LIN {X 0,Y 467.704,Z 292.228,A -85,B 0,C 180,E1 -7476.035,E2 -7476.035} C_VEL
LIN {X 0,Y 467.665,Z 292.229,A -85,B 0,C 180,E1 -7478.64,E2 -7478.64} C_VEL
LIN {X 0,Y 467.684,Z 292.329,A -85,B 0,C 180,E1 -7481.125,E2 -7481.125} C_VEL
LIN {X 0,Y 468.727,Z 299.708,A -85,B 0,C 180,E1 -7482.725,E2 -7482.725} C_VEL
LIN {X 0,Y 468.456,Z 310.96,A -85,B 0,C 180,E1 -7485.05,E2 -7485.05} C_VEL
LIN {X 0,Y 471.306,Z 325.447,A -85,B 0,C 180,E1 -7485.4,E2 -7485.4} C_VEL
LIN {X 0,Y 470.52,Z 418.247,A -85,B 0,C 180,E1 -7486.862,E2 -7486.862} C_VEL
LIN {X 0,Y 470.256,Z 431.761,A -85,B 0,C 180,E1 -7487.255,E2 -7487.255} C_VEL
LIN {X 0,Y 469.928,Z 444.22,A -85,B 0,C 180,E1 -7487.793,E2 -7487.793} C_VEL
LIN {X 0,Y 469.506,Z 455.23,A -85,B 0,C 180,E1 -7488.43,E2 -7488.43} C_VEL
LIN {X 0,Y 469.027,Z 466.456,A -85,B 0,C 180,E1 -7489.264,E2 -7489.264} C_VEL
LIN {X 0,Y 468.47,Z 477.517,A -85,B 0,C 180,E1 -7490.295,E2 -7490.295} C_VEL
LIN {X 0,Y 468.012,Z 487.034,A -85,B 0,C 180,E1 -7491.402,E2 -7491.402} C_VEL
LIN {X 0,Y 467.679,Z 494.909,A -85,B 0,C 180,E1 -7492.527,E2 -7492.527} C_VEL
LIN {X 0,Y 467.319,Z 502.972,A -85,B 0,C 180,E1 -7493.952,E2 -7493.952} C_VEL
LIN {X 0,Y 467.082,Z 508.521,A -85,B 0,C 180,E1 -7495.183,E2 -7495.183} C_VEL
LIN {X 0,Y 466.913,Z 512.769,A -85,B 0,C 180,E1 -7496.357,E2 -7496.357} C_VEL
LIN {X 0,Y 466.762,Z 516.837,A -85,B 0,C 180,E1 -7497.819,E2 -7497.819} C_VEL
LIN {X 0,Y 466.632,Z 519.377,A -85,B 0,C 180,E1 -7499.126,E2 -7499.126} C_VEL
LIN {X 0,Y 466.562,Z 521.275,A -85,B 0,C 180,E1 -7500.838,E2 -7500.838} C_VEL
LIN {X 0,Y 466.549,Z 521.623,A -85,B 0,C 180,E1 -7502.48,E2 -7502.48} C_VEL
LIN {X 0,Y 466.552,Z 520.636,A -85,B 0,C 180,E1 -7504.054,E2 -7504.054} C_VEL
LIN {X 0,Y 466.699,Z 518.356,A -85,B 0,C 180,E1 -7505.591,E2 -7505.591} C_VEL
LIN {X 0,Y 466.821,Z 514.889,A -85,B 0,C 180,E1 -7507.068,E2 -7507.068} C_VEL
LIN {X 0,Y 467.024,Z 510.213,A -85,B 0,C 180,E1 -7508.508,E2 -7508.508} C_VEL
LIN {X 0,Y 467.265,Z 504.294,A -85,B 0,C 180,E1 -7509.908,E2 -7509.908} C_VEL
LIN {X 0,Y 467.591,Z 496.918,A -85,B 0,C 180,E1 -7511.278,E2 -7511.278} C_VEL
LIN {X 0,Y 468.015,Z 488.675,A -85,B 0,C 180,E1 -7512.505,E2 -7512.505} C_VEL
LIN {X 0,Y 468.474,Z 479.399,A -85,B 0,C 180,E1 -7513.629,E2 -7513.629} C_VEL
LIN {X 0,Y 468.998,Z 468.987,A -85,B 0,C 180,E1 -7514.648,E2 -7514.648} C_VEL
LIN {X 0,Y 469.505,Z 457.587,A -85,B 0,C 180,E1 -7515.532,E2 -7515.532} C_VEL
LIN {X 0,Y 469.927,Z 445.273,A -85,B 0,C 180,E1 -7516.277,E2 -7516.277} C_VEL
LIN {X 0,Y 470.301,Z 432.788,A -85,B 0,C 180,E1 -7516.829,E2 -7516.829} C_VEL
LIN {X 0,Y 470.561,Z 419.847,A -85,B 0,C 180,E1 -7517.218,E2 -7517.218} C_VEL
LIN {X 0,Y 470.874,Z 388.179,A -85,B 0,C 180,E1 -7517.741,E2 -7517.741} C_VEL
LIN {X 0,Y 471.357,Z 325.273,A -85,B 0,C 180,E1 -7518.725,E2 -7518.725} C_VEL
LIN {X 0,Y 468.506,Z 310.615,A -85,B 0,C 180,E1 -7519.089,E2 -7519.089} C_VEL
LIN {X 0,Y 468.614,Z 298.408,A -85,B 0,C 180,E1 -7521.344,E2 -7521.344} C_VEL
LIN {X 0,Y 467.552,Z 292.248,A -85,B 0,C 180,E1 -7522.545,E2 -7522.545} C_VEL
LIN {X 0,Y 467.55,Z 292.246,A -85,B 0,C 180,E1 -7525.754,E2 -7525.754} C_VEL
LIN {X 0,Y 467.529,Z 292.247,A -85,B 0,C 180,E1 -7528.951,E2 -7528.951} C_VEL
LIN {X 0,Y 467.601,Z 292.244,A -85,B 0,C 180,E1 -7532.456,E2 -7532.456} C_VEL
LIN {X 0,Y 467.557,Z 292.245,A -85,B 0,C 180,E1 -7535.11,E2 -7535.11} C_VEL
LIN {X 0,Y 467.485,Z 292.255,A -85,B 0,C 180,E1 -7537.924,E2 -7537.924} C_VEL
LIN {X 0,Y 467.573,Z 292.244,A -85,B 0,C 180,E1 -7540.69,E2 -7540.69} C_VEL
LIN {X 0,Y 467.597,Z 292.237,A -85,B 0,C 180,E1 -7544.113,E2 -7544.113} C_VEL
LIN {X 0,Y 467.601,Z 292.235,A -85,B 0,C 180,E1 -7547.641,E2 -7547.641} C_VEL
LIN {X 0,Y 467.613,Z 292.236,A -85,B 0,C 180,E1 -7550.484,E2 -7550.484} C_VEL
LIN {X 0,Y 467.646,Z 292.232,A -85,B 0,C 180,E1 -7553.095,E2 -7553.095} C_VEL
LIN {X 0,Y 467.67,Z 292.231,A -85,B 0,C 180,E1 -7554.827,E2 -7554.827} C_VEL
LIN {X 0,Y 467.811,Z 292.209,A -85,B 0,C 180,E1 -7557.417,E2 -7557.417} C_VEL
LIN {X 0,Y 467.776,Z 292.217,A -85,B 0,C 180,E1 -7560.861,E2 -7560.861} C_VEL
LIN {X 0,Y 467.813,Z 292.212,A -85,B 0,C 180,E1 -7562.583,E2 -7562.583} C_VEL
LIN {X 0,Y 467.699,Z 292.222,A -85,B 0,C 180,E1 -7566.038,E2 -7566.038} C_VEL
LIN {X 0,Y 467.636,Z 292.229,A -85,B 0,C 180,E1 -7568.644,E2 -7568.644} C_VEL
LIN {X 0,Y 467.646,Z 292.224,A -85,B 0,C 180,E1 -7572.146,E2 -7572.146} C_VEL
LIN {X 0,Y 467.617,Z 292.228,A -85,B 0,C 180,E1 -7575.895,E2 -7575.895} C_VEL
LIN {X 0,Y 467.575,Z 292.24,A -85,B 0,C 180,E1 -7579.31,E2 -7579.31} C_VEL
LIN {X 0,Y 467.532,Z 292.242,A -85,B 0,C 180,E1 -7582.074,E2 -7582.074} C_VEL
LIN {X 0,Y 467.575,Z 292.235,A -85,B 0,C 180,E1 -7584.889,E2 -7584.889} C_VEL
LIN {X 0,Y 467.584,Z 292.236,A -85,B 0,C 180,E1 -7587.771,E2 -7587.771} C_VEL
LIN {X 0,Y 467.531,Z 292.246,A -85,B 0,C 180,E1 -7591.049,E2 -7591.049} C_VEL
LIN {X 0,Y 467.55,Z 292.24,A -85,B 0,C 180,E1 -7594.246,E2 -7594.246} C_VEL
LIN {X 0,Y 467.524,Z 292.248,A -85,B 0,C 180,E1 -7597.192,E2 -7597.192} C_VEL
LIN {X 0,Y 467.579,Z 292.241,A -85,B 0,C 180,E1 -7599.963,E2 -7599.963} C_VEL
LIN {X 0,Y 467.586,Z 292.239,A -85,B 0,C 180,E1 -7602.575,E2 -7602.575} C_VEL
LIN {X 0,Y 467.544,Z 292.247,A -85,B 0,C 180,E1 -7606.181,E2 -7606.181} C_VEL
LIN {X 0,Y 467.563,Z 292.241,A -85,B 0,C 180,E1 -7608.726,E2 -7608.726} C_VEL
LIN {X 0,Y 467.555,Z 292.245,A -85,B 0,C 180,E1 -7611.411,E2 -7611.411} C_VEL
LIN {X 0,Y 467.541,Z 292.247,A -85,B 0,C 180,E1 -7614.264,E2 -7614.264} C_VEL
LIN {X 0,Y 467.563,Z 292.245,A -85,B 0,C 180,E1 -7617.325,E2 -7617.325} C_VEL
LIN {X 0,Y 467.562,Z 292.245,A -85,B 0,C 180,E1 -7620.67,E2 -7620.67} C_VEL
LIN {X 0,Y 467.614,Z 292.24,A -85,B 0,C 180,E1 -7623.686,E2 -7623.686} C_VEL
LIN {X 0,Y 467.64,Z 292.332,A -85,B 0,C 180,E1 -7624.137,E2 -7624.137} C_VEL
LIN {X 0,Y 469.709,Z 303.354,A -85,B 0,C 180,E1 -7626.177,E2 -7626.177} C_VEL
LIN {X 0,Y 469.179,Z 319.417,A -85,B 0,C 180,E1 -7628.935,E2 -7628.935} C_VEL
LIN {X 0,Y 468.465,Z 338.052,A -85,B 0,C 180,E1 -7632.093,E2 -7632.093} C_VEL
LIN {X 0,Y 468.269,Z 343.322,A -85,B 0,C 180,E1 -7632.962,E2 -7632.962} C_VEL
LIN {X 0,Y 471.212,Z 363.176,A -85,B 0,C 180,E1 -7633.389,E2 -7633.389} C_VEL
LIN {X 0,Y 470.443,Z 452.18,A -85,B 0,C 180,E1 -7634.793,E2 -7634.793} C_VEL
LIN {X 0,Y 470.061,Z 466.055,A -85,B 0,C 180,E1 -7635.196,E2 -7635.196} C_VEL
LIN {X 0,Y 469.561,Z 479.027,A -85,B 0,C 180,E1 -7635.762,E2 -7635.762} C_VEL
LIN {X 0,Y 469.134,Z 490.835,A -85,B 0,C 180,E1 -7636.467,E2 -7636.467} C_VEL
LIN {X 0,Y 468.58,Z 502.825,A -85,B 0,C 180,E1 -7637.383,E2 -7637.383} C_VEL
LIN {X 0,Y 468.157,Z 512.507,A -85,B 0,C 180,E1 -7638.311,E2 -7638.311} C_VEL
LIN {X 0,Y 467.69,Z 521.747,A -85,B 0,C 180,E1 -7639.396,E2 -7639.396} C_VEL
LIN {X 0,Y 467.274,Z 530.751,A -85,B 0,C 180,E1 -7640.699,E2 -7640.699} C_VEL
LIN {X 0,Y 467.006,Z 538.009,A -85,B 0,C 180,E1 -7642.002,E2 -7642.002} C_VEL
LIN {X 0,Y 466.851,Z 542.909,A -85,B 0,C 180,E1 -7643.086,E2 -7643.086} C_VEL
LIN {X 0,Y 466.76,Z 547.675,A -85,B 0,C 180,E1 -7644.387,E2 -7644.387} C_VEL
LIN {X 0,Y 466.646,Z 551.315,A -85,B 0,C 180,E1 -7645.684,E2 -7645.684} C_VEL
LIN {X 0,Y 466.689,Z 553.198,A -85,B 0,C 180,E1 -7646.55,E2 -7646.55} C_VEL
LIN {X 0,Y 466.661,Z 554.607,A -85,B 0,C 180,E1 -7647.413,E2 -7647.413} C_VEL
LIN {X 0,Y 466.619,Z 556.232,A -85,B 0,C 180,E1 -7649.14,E2 -7649.14} C_VEL
LIN {X 0,Y 466.6,Z 556.451,A -85,B 0,C 180,E1 -7650.003,E2 -7650.003} C_VEL
LIN {X 0,Y 466.619,Z 556.236,A -85,B 0,C 180,E1 -7650.866,E2 -7650.866} C_VEL
LIN {X 0,Y 466.662,Z 554.629,A -85,B 0,C 180,E1 -7652.592,E2 -7652.592} C_VEL
LIN {X 0,Y 466.69,Z 553.223,A -85,B 0,C 180,E1 -7653.456,E2 -7653.456} C_VEL
LIN {X 0,Y 466.69,Z 550.267,A -85,B 0,C 180,E1 -7654.753,E2 -7654.753} C_VEL
LIN {X 0,Y 466.752,Z 546.264,A -85,B 0,C 180,E1 -7656.053,E2 -7656.053} C_VEL
LIN {X 0,Y 466.943,Z 540.102,A -85,B 0,C 180,E1 -7657.57,E2 -7657.57} C_VEL
LIN {X 0,Y 467.167,Z 533.373,A -85,B 0,C 180,E1 -7658.873,E2 -7658.873} C_VEL
LIN {X 0,Y 467.505,Z 525.026,A -85,B 0,C 180,E1 -7660.176,E2 -7660.176} C_VEL
LIN {X 0,Y 467.954,Z 516.447,A -85,B 0,C 180,E1 -7661.261,E2 -7661.261} C_VEL
LIN {X 0,Y 468.472,Z 506.349,A -85,B 0,C 180,E1 -7662.3,E2 -7662.3} C_VEL
LIN {X 0,Y 468.906,Z 495.369,A -85,B 0,C 180,E1 -7663.215,E2 -7663.215} C_VEL
LIN {X 0,Y 469.392,Z 483.818,A -85,B 0,C 180,E1 -7663.973,E2 -7663.973} C_VEL
LIN {X 0,Y 469.832,Z 471.84,A -85,B 0,C 180,E1 -7664.568,E2 -7664.568} C_VEL
LIN {X 0,Y 470.277,Z 458.915,A -85,B 0,C 180,E1 -7665.024,E2 -7665.024} C_VEL
LIN {X 0,Y 470.546,Z 445.237,A -85,B 0,C 180,E1 -7665.32,E2 -7665.32} C_VEL
LIN {X 0,Y 471.139,Z 362.545,A -85,B 0,C 180,E1 -7666.605,E2 -7666.605} C_VEL
LIN {X 0,Y 468.314,Z 343.69,A -85,B 0,C 180,E1 -7667.018,E2 -7667.018} C_VEL
LIN {X 0,Y 469.052,Z 325.465,A -85,B 0,C 180,E1 -7670.16,E2 -7670.16} C_VEL
LIN {X 0,Y 469.878,Z 307.217,A -85,B 0,C 180,E1 -7673.352,E2 -7673.352} C_VEL
LIN {X 0,Y 469.713,Z 302.985,A -85,B 0,C 180,E1 -7674.118,E2 -7674.118} C_VEL
LIN {X 0,Y 467.659,Z 292.234,A -85,B 0,C 180,E1 -7676.197,E2 -7676.197} C_VEL
LIN {X 0,Y 467.573,Z 292.242,A -85,B 0,C 180,E1 -7679.333,E2 -7679.333} C_VEL
LIN {X 0,Y 467.585,Z 292.237,A -85,B 0,C 180,E1 -7682.679,E2 -7682.679} C_VEL
LIN {X 0,Y 467.563,Z 292.241,A -85,B 0,C 180,E1 -7685.739,E2 -7685.739} C_VEL
LIN {X 0,Y 467.562,Z 292.238,A -85,B 0,C 180,E1 -7689.147,E2 -7689.147} C_VEL
LIN {X 0,Y 467.588,Z 292.241,A -85,B 0,C 180,E1 -7692.567,E2 -7692.567} C_VEL
LIN {X 0,Y 467.566,Z 292.239,A -85,B 0,C 180,E1 -7695.052,E2 -7695.052} C_VEL
LIN {X 0,Y 467.589,Z 292.235,A -85,B 0,C 180,E1 -7697.44,E2 -7697.44} C_VEL
LIN {X 0,Y 467.58,Z 292.24,A -85,B 0,C 180,E1 -7700.855,E2 -7700.855} C_VEL
LIN {X 0,Y 467.559,Z 292.242,A -85,B 0,C 180,E1 -7704.26,E2 -7704.26} C_VEL
LIN {X 0,Y 467.579,Z 292.237,A -85,B 0,C 180,E1 -7707.321,E2 -7707.321} C_VEL
LIN {X 0,Y 467.567,Z 292.245,A -85,B 0,C 180,E1 -7710.667,E2 -7710.667} C_VEL
LIN {X 0,Y 467.611,Z 292.236,A -85,B 0,C 180,E1 -7713.199,E2 -7713.199} C_VEL
LIN {X 0,Y 467.587,Z 292.238,A -85,B 0,C 180,E1 -7716.468,E2 -7716.468} C_VEL
LIN {X 0,Y 467.615,Z 292.232,A -85,B 0,C 180,E1 -7719.777,E2 -7719.777} C_VEL
LIN {X 0,Y 467.598,Z 292.235,A -85,B 0,C 180,E1 -7722.506,E2 -7722.506} C_VEL
LIN {X 0,Y 467.597,Z 292.242,A -85,B 0,C 180,E1 -7725.196,E2 -7725.196} C_VEL
LIN {X 0,Y 467.647,Z 292.229,A -85,B 0,C 180,E1 -7727.854,E2 -7727.854} C_VEL
LIN {X 0,Y 467.672,Z 292.232,A -85,B 0,C 180,E1 -7731.357,E2 -7731.357} C_VEL
LIN {X 0,Y 467.723,Z 292.219,A -85,B 0,C 180,E1 -7733.962,E2 -7733.962} C_VEL
LIN {X 0,Y 467.847,Z 292.212,A -85,B 0,C 180,E1 -7737.417,E2 -7737.417} C_VEL
LIN {X 0,Y 467.866,Z 292.202,A -85,B 0,C 180,E1 -7740,E2 -7740} C_VEL
LIN {X 0,Y 467.846,Z 292.203,A -85,B 0,C 180,E1 -7742.583,E2 -7742.583} C_VEL
LIN {X 0,Y 467.708,Z 292.223,A -85,B 0,C 180,E1 -7746.038,E2 -7746.038} C_VEL
LIN {X 0,Y 467.659,Z 292.226,A -85,B 0,C 180,E1 -7748.643,E2 -7748.643} C_VEL
LIN {X 0,Y 467.646,Z 292.231,A -85,B 0,C 180,E1 -7752.146,E2 -7752.146} C_VEL
LIN {X 0,Y 467.64,Z 292.237,A -85,B 0,C 180,E1 -7755.884,E2 -7755.884} C_VEL
LIN {X 0,Y 467.612,Z 292.233,A -85,B 0,C 180,E1 -7759.308,E2 -7759.308} C_VEL
LIN {X 0,Y 467.522,Z 292.251,A -85,B 0,C 180,E1 -7762.075,E2 -7762.075} C_VEL
LIN {X 0,Y 467.548,Z 292.24,A -85,B 0,C 180,E1 -7764.891,E2 -7764.891} C_VEL
LIN {X 0,Y 467.537,Z 292.245,A -85,B 0,C 180,E1 -7767.774,E2 -7767.774} C_VEL
LIN {X 0,Y 467.543,Z 292.241,A -85,B 0,C 180,E1 -7771.041,E2 -7771.041} C_VEL
LIN {X 0,Y 467.571,Z 292.245,A -85,B 0,C 180,E1 -7774.24,E2 -7774.24} C_VEL
LIN {X 0,Y 467.51,Z 292.245,A -85,B 0,C 180,E1 -7777.181,E2 -7777.181} C_VEL
LIN {X 0,Y 467.535,Z 292.248,A -85,B 0,C 180,E1 -7780.269,E2 -7780.269} C_VEL
LIN {X 0,Y 467.515,Z 292.252,A -85,B 0,C 180,E1 -7782.569,E2 -7782.569} C_VEL
LIN {X 0,Y 467.552,Z 292.242,A -85,B 0,C 180,E1 -7785.051,E2 -7785.051} C_VEL
LIN {X 0,Y 467.55,Z 292.247,A -85,B 0,C 180,E1 -7788.727,E2 -7788.727} C_VEL
LIN {X 0,Y 467.532,Z 292.242,A -85,B 0,C 180,E1 -7791.952,E2 -7791.952} C_VEL
LIN {X 0,Y 467.489,Z 292.251,A -85,B 0,C 180,E1 -7795.16,E2 -7795.16} C_VEL
LIN {X 0,Y 467.543,Z 292.242,A -85,B 0,C 180,E1 -7798.256,E2 -7798.256} C_VEL
LIN {X 0,Y 467.528,Z 292.247,A -85,B 0,C 180,E1 -7801.246,E2 -7801.246} C_VEL
LIN {X 0,Y 467.563,Z 292.239,A -85,B 0,C 180,E1 -7804.405,E2 -7804.405} C_VEL
LIN {X 0,Y 467.577,Z 292.244,A -85,B 0,C 180,E1 -7806.995,E2 -7806.995} C_VEL
LIN {X 0,Y 467.623,Z 292.232,A -85,B 0,C 180,E1 -7809.776,E2 -7809.776} C_VEL
LIN {X 0,Y 467.589,Z 292.235,A -85,B 0,C 180,E1 -7812.504,E2 -7812.504} C_VEL
LIN {X 0,Y 467.594,Z 292.239,A -85,B 0,C 180,E1 -7815.403,E2 -7815.403} C_VEL
LIN {X 0,Y 466.923,Z 292.32,A -85,B 0,C 180,E1 -7816.123,E2 -7816.123} C_VEL
LIN {X 0,Y 464.083,Z 292.68,A -85,B 0,C 180,E1 -7817.291,E2 -7817.291} C_VEL
LIN {X 0,Y 461.685,Z 292.974,A -85,B 0,C 180,E1 -7818.233,E2 -7818.233} C_VEL
LIN {X 0,Y 460.655,Z 293.102,A -85,B 0,C 180,E1 -7818.961,E2 -7818.961} C_VEL
LIN {X 0,Y 460.57,Z 293.114,A -85,B 0,C 180,E1 -7819.208,E2 -7819.208} C_VEL
LIN {X 0,Y 460.668,Z 293.097,A -85,B 0,C 180,E1 -7822.591,E2 -7822.591} C_VEL
LIN {X 0,Y 460.678,Z 293.096,A -85,B 0,C 180,E1 -7824.746,E2 -7824.746} C_VEL
LIN {X 0,Y 460.759,Z 293.091,A -85,B 0,C 180,E1 -7827.375,E2 -7827.375} C_VEL
LIN {X 0,Y 460.821,Z 293.081,A -85,B 0,C 180,E1 -7829.997,E2 -7829.997} C_VEL
LIN {X 0,Y 460.76,Z 293.085,A -85,B 0,C 180,E1 -7832.62,E2 -7832.62} C_VEL
LIN {X 0,Y 460.669,Z 293.103,A -85,B 0,C 180,E1 -7836.127,E2 -7836.127} C_VEL
LIN {X 0,Y 460.615,Z 293.107,A -85,B 0,C 180,E1 -7838.773,E2 -7838.773} C_VEL
LIN {X 0,Y 460.613,Z 293.147,A -85,B 0,C 180,E1 -7840.936,E2 -7840.936} C_VEL
LIN {X 0,Y 461.761,Z 300.65,A -85,B 0,C 180,E1 -7842.59,E2 -7842.59} C_VEL
LIN {X 0,Y 461.491,Z 311.259,A -85,B 0,C 180,E1 -7844.803,E2 -7844.803} C_VEL
LIN {X 0,Y 464.534,Z 327.145,A -85,B 0,C 180,E1 -7845.18,E2 -7845.18} C_VEL
LIN {X 0,Y 463.635,Z 418.904,A -85,B 0,C 180,E1 -7846.65,E2 -7846.65} C_VEL
LIN {X 0,Y 463.391,Z 432.539,A -85,B 0,C 180,E1 -7847.059,E2 -7847.059} C_VEL
LIN {X 0,Y 463.054,Z 444.473,A -85,B 0,C 180,E1 -7847.586,E2 -7847.586} C_VEL
LIN {X 0,Y 462.588,Z 455.843,A -85,B 0,C 180,E1 -7848.257,E2 -7848.257} C_VEL
LIN {X 0,Y 462.039,Z 467.632,A -85,B 0,C 180,E1 -7849.156,E2 -7849.156} C_VEL
LIN {X 0,Y 461.497,Z 478.025,A -85,B 0,C 180,E1 -7850.15,E2 -7850.15} C_VEL
LIN {X 0,Y 461.037,Z 487.092,A -85,B 0,C 180,E1 -7851.221,E2 -7851.221} C_VEL
LIN {X 0,Y 460.665,Z 495.329,A -85,B 0,C 180,E1 -7852.416,E2 -7852.416} C_VEL
LIN {X 0,Y 460.328,Z 502.267,A -85,B 0,C 180,E1 -7853.645,E2 -7853.645} C_VEL
LIN {X 0,Y 460.043,Z 507.767,A -85,B 0,C 180,E1 -7854.837,E2 -7854.837} C_VEL
LIN {X 0,Y 459.857,Z 513.12,A -85,B 0,C 180,E1 -7856.304,E2 -7856.304} C_VEL
LIN {X 0,Y 459.683,Z 516.546,A -85,B 0,C 180,E1 -7857.532,E2 -7857.532} C_VEL
LIN {X 0,Y 459.595,Z 518.224,A -85,B 0,C 180,E1 -7858.292,E2 -7858.292} C_VEL
LIN {X 0,Y 459.521,Z 520.017,A -85,B 0,C 180,E1 -7859.335,E2 -7859.335} C_VEL
LIN {X 0,Y 459.45,Z 521.671,A -85,B 0,C 180,E1 -7861.062,E2 -7861.062} C_VEL
LIN {X 0,Y 459.437,Z 521.849,A -85,B 0,C 180,E1 -7862.718,E2 -7862.718} C_VEL
LIN {X 0,Y 459.481,Z 520.459,A -85,B 0,C 180,E1 -7864.461,E2 -7864.461} C_VEL
LIN {X 0,Y 459.647,Z 518.184,A -85,B 0,C 180,E1 -7865.868,E2 -7865.868} C_VEL
LIN {X 0,Y 459.775,Z 514.575,A -85,B 0,C 180,E1 -7867.358,E2 -7867.358} C_VEL
LIN {X 0,Y 460.026,Z 509.729,A -85,B 0,C 180,E1 -7868.817,E2 -7868.817} C_VEL
LIN {X 0,Y 460.261,Z 503.628,A -85,B 0,C 180,E1 -7870.228,E2 -7870.228} C_VEL
LIN {X 0,Y 460.634,Z 496.009,A -85,B 0,C 180,E1 -7871.616,E2 -7871.616} C_VEL
LIN {X 0,Y 461.126,Z 487.15,A -85,B 0,C 180,E1 -7872.912,E2 -7872.912} C_VEL
LIN {X 0,Y 461.667,Z 477.05,A -85,B 0,C 180,E1 -7874.089,E2 -7874.089} C_VEL
LIN {X 0,Y 462.21,Z 465.78,A -85,B 0,C 180,E1 -7875.141,E2 -7875.141} C_VEL
LIN {X 0,Y 462.718,Z 454.964,A -85,B 0,C 180,E1 -7875.938,E2 -7875.938} C_VEL
LIN {X 0,Y 463.137,Z 443.723,A -85,B 0,C 180,E1 -7876.586,E2 -7876.586} C_VEL
LIN {X 0,Y 463.558,Z 430.282,A -85,B 0,C 180,E1 -7877.154,E2 -7877.154} C_VEL
LIN {X 0,Y 463.804,Z 417.667,A -85,B 0,C 180,E1 -7877.506,E2 -7877.506} C_VEL
LIN {X 0,Y 464.631,Z 326.727,A -85,B 0,C 180,E1 -7878.962,E2 -7878.962} C_VEL
LIN {X 0,Y 461.585,Z 310.91,A -85,B 0,C 180,E1 -7879.352,E2 -7879.352} C_VEL
LIN {X 0,Y 461.605,Z 298.605,A -85,B 0,C 180,E1 -7881.653,E2 -7881.653} C_VEL
LIN {X 0,Y 460.532,Z 293.121,A -85,B 0,C 180,E1 -7882.774,E2 -7882.774} C_VEL
LIN {X 0,Y 460.509,Z 293.123,A -85,B 0,C 180,E1 -7885.62,E2 -7885.62} C_VEL
LIN {X 0,Y 460.495,Z 293.125,A -85,B 0,C 180,E1 -7888.741,E2 -7888.741} C_VEL
LIN {X 0,Y 460.545,Z 293.123,A -85,B 0,C 180,E1 -7892.249,E2 -7892.249} C_VEL
LIN {X 0,Y 460.513,Z 293.126,A -85,B 0,C 180,E1 -7894.703,E2 -7894.703} C_VEL
LIN {X 0,Y 460.462,Z 293.128,A -85,B 0,C 180,E1 -7897.569,E2 -7897.569} C_VEL
LIN {X 0,Y 460.519,Z 293.126,A -85,B 0,C 180,E1 -7900.382,E2 -7900.382} C_VEL
LIN {X 0,Y 460.514,Z 293.119,A -85,B 0,C 180,E1 -7903.144,E2 -7903.144} C_VEL
LIN {X 0,Y 460.501,Z 293.12,A -85,B 0,C 180,E1 -7905.866,E2 -7905.866} C_VEL
LIN {X 0,Y 460.56,Z 293.119,A -85,B 0,C 180,E1 -7908.558,E2 -7908.558} C_VEL
LIN {X 0,Y 460.642,Z 293.102,A -85,B 0,C 180,E1 -7912.108,E2 -7912.108} C_VEL
LIN {X 0,Y 460.642,Z 293.108,A -85,B 0,C 180,E1 -7914.748,E2 -7914.748} C_VEL
LIN {X 0,Y 460.777,Z 293.086,A -85,B 0,C 180,E1 -7917.377,E2 -7917.377} C_VEL
LIN {X 0,Y 460.796,Z 293.077,A -85,B 0,C 180,E1 -7920,E2 -7920} C_VEL
LIN {X 0,Y 460.779,Z 293.088,A -85,B 0,C 180,E1 -7922.623,E2 -7922.623} C_VEL
LIN {X 0,Y 460.663,Z 293.099,A -85,B 0,C 180,E1 -7926.131,E2 -7926.131} C_VEL
LIN {X 0,Y 460.583,Z 293.109,A -85,B 0,C 180,E1 -7928.777,E2 -7928.777} C_VEL
LIN {X 0,Y 460.606,Z 293.101,A -85,B 0,C 180,E1 -7932.334,E2 -7932.334} C_VEL
LIN {X 0,Y 460.572,Z 293.105,A -85,B 0,C 180,E1 -7936.009,E2 -7936.009} C_VEL
LIN {X 0,Y 460.521,Z 293.115,A -85,B 0,C 180,E1 -7939.618,E2 -7939.618} C_VEL
LIN {X 0,Y 460.495,Z 293.118,A -85,B 0,C 180,E1 -7942.43,E2 -7942.43} C_VEL
LIN {X 0,Y 460.54,Z 293.115,A -85,B 0,C 180,E1 -7945.809,E2 -7945.809} C_VEL
LIN {X 0,Y 460.515,Z 293.113,A -85,B 0,C 180,E1 -7948.236,E2 -7948.236} C_VEL
LIN {X 0,Y 460.483,Z 293.126,A -85,B 0,C 180,E1 -7951.287,E2 -7951.287} C_VEL
LIN {X 0,Y 460.496,Z 293.119,A -85,B 0,C 180,E1 -7954.51,E2 -7954.51} C_VEL
LIN {X 0,Y 460.506,Z 293.124,A -85,B 0,C 180,E1 -7957.623,E2 -7957.623} C_VEL
LIN {X 0,Y 460.531,Z 293.117,A -85,B 0,C 180,E1 -7960.277,E2 -7960.277} C_VEL
LIN {X 0,Y 460.492,Z 293.127,A -85,B 0,C 180,E1 -7963.376,E2 -7963.376} C_VEL
LIN {X 0,Y 460.495,Z 293.123,A -85,B 0,C 180,E1 -7966.632,E2 -7966.632} C_VEL
LIN {X 0,Y 460.537,Z 293.123,A -85,B 0,C 180,E1 -7969.732,E2 -7969.732} C_VEL
LIN {X 0,Y 460.506,Z 293.12,A -85,B 0,C 180,E1 -7972.523,E2 -7972.523} C_VEL
LIN {X 0,Y 460.528,Z 293.123,A -85,B 0,C 180,E1 -7975.628,E2 -7975.628} C_VEL
LIN {X 0,Y 460.518,Z 293.123,A -85,B 0,C 180,E1 -7978.749,E2 -7978.749} C_VEL
LIN {X 0,Y 460.543,Z 293.121,A -85,B 0,C 180,E1 -7981.772,E2 -7981.772} C_VEL
LIN {X 0,Y 460.595,Z 293.307,A -85,B 0,C 180,E1 -7983.938,E2 -7983.938} C_VEL
LIN {X 0,Y 462.755,Z 304.422,A -85,B 0,C 180,E1 -7986.035,E2 -7986.035} C_VEL
LIN {X 0,Y 462.223,Z 320.485,A -85,B 0,C 180,E1 -7988.836,E2 -7988.836} C_VEL
LIN {X 0,Y 461.45,Z 339.136,A -85,B 0,C 180,E1 -7992.041,E2 -7992.041} C_VEL
LIN {X 0,Y 461.299,Z 342.87,A -85,B 0,C 180,E1 -7992.678,E2 -7992.678} C_VEL
LIN {X 0,Y 464.398,Z 363.338,A -85,B 0,C 180,E1 -7993.14,E2 -7993.14} C_VEL
LIN {X 0,Y 463.613,Z 452.008,A -85,B 0,C 180,E1 -7994.564,E2 -7994.564} C_VEL
LIN {X 0,Y 463.212,Z 465.843,A -85,B 0,C 180,E1 -7994.972,E2 -7994.972} C_VEL
LIN {X 0,Y 462.661,Z 478.791,A -85,B 0,C 180,E1 -7995.545,E2 -7995.545} C_VEL
LIN {X 0,Y 462.202,Z 490.591,A -85,B 0,C 180,E1 -7996.26,E2 -7996.26} C_VEL
LIN {X 0,Y 461.685,Z 501.803,A -85,B 0,C 180,E1 -7997.125,E2 -7997.125} C_VEL
LIN {X 0,Y 461.182,Z 512.255,A -85,B 0,C 180,E1 -7998.132,E2 -7998.132} C_VEL
LIN {X 0,Y 460.655,Z 521.492,A -85,B 0,C 180,E1 -7999.232,E2 -7999.232} C_VEL
LIN {X 0,Y 460.241,Z 530.496,A -85,B 0,C 180,E1 -8000.555,E2 -8000.555} C_VEL
LIN {X 0,Y 459.947,Z 537.749,A -85,B 0,C 180,E1 -8001.878,E2 -8001.878} C_VEL
LIN {X 0,Y 459.74,Z 543.825,A -85,B 0,C 180,E1 -8003.276,E2 -8003.276} C_VEL
LIN {X 0,Y 459.649,Z 548.735,A -85,B 0,C 180,E1 -8004.74,E2 -8004.74} C_VEL
LIN {X 0,Y 459.564,Z 551.051,A -85,B 0,C 180,E1 -8005.618,E2 -8005.618} C_VEL
LIN {X 0,Y 459.584,Z 552.932,A -85,B 0,C 180,E1 -8006.496,E2 -8006.496} C_VEL
LIN {X 0,Y 459.583,Z 554.343,A -85,B 0,C 180,E1 -8007.374,E2 -8007.374} C_VEL
LIN {X 0,Y 459.552,Z 555.968,A -85,B 0,C 180,E1 -8009.127,E2 -8009.127} C_VEL
LIN {X 0,Y 459.532,Z 556.188,A -85,B 0,C 180,E1 -8010.003,E2 -8010.003} C_VEL
LIN {X 0,Y 459.552,Z 555.972,A -85,B 0,C 180,E1 -8010.879,E2 -8010.879} C_VEL
LIN {X 0,Y 459.585,Z 554.364,A -85,B 0,C 180,E1 -8012.632,E2 -8012.632} C_VEL
LIN {X 0,Y 459.586,Z 552.954,A -85,B 0,C 180,E1 -8013.509,E2 -8013.509} C_VEL
LIN {X 0,Y 459.618,Z 549.997,A -85,B 0,C 180,E1 -8014.827,E2 -8014.827} C_VEL
LIN {X 0,Y 459.716,Z 544.945,A -85,B 0,C 180,E1 -8016.433,E2 -8016.433} C_VEL
LIN {X 0,Y 459.893,Z 538.801,A -85,B 0,C 180,E1 -8017.908,E2 -8017.908} C_VEL
LIN {X 0,Y 460.177,Z 531.835,A -85,B 0,C 180,E1 -8019.23,E2 -8019.23} C_VEL
LIN {X 0,Y 460.563,Z 523.1,A -85,B 0,C 180,E1 -8020.553,E2 -8020.553} C_VEL
LIN {X 0,Y 461.065,Z 514.156,A -85,B 0,C 180,E1 -8021.654,E2 -8021.654} C_VEL
LIN {X 0,Y 461.565,Z 503.409,A -85,B 0,C 180,E1 -8022.731,E2 -8022.731} C_VEL
LIN {X 0,Y 462.096,Z 491.943,A -85,B 0,C 180,E1 -8023.637,E2 -8023.637} C_VEL
LIN {X 0,Y 462.661,Z 479.417,A -85,B 0,C 180,E1 -8024.405,E2 -8024.405} C_VEL
LIN {X 0,Y 463.135,Z 466.639,A -85,B 0,C 180,E1 -8024.98,E2 -8024.98} C_VEL
LIN {X 0,Y 463.526,Z 453.049,A -85,B 0,C 180,E1 -8025.389,E2 -8025.389} C_VEL
LIN {X 0,Y 464.013,Z 411.749,A -85,B 0,C 180,E1 -8026.063,E2 -8026.063} C_VEL
LIN {X 0,Y 464.242,Z 362.685,A -85,B 0,C 180,E1 -8026.845,E2 -8026.845} C_VEL
LIN {X 0,Y 461.307,Z 343.464,A -85,B 0,C 180,E1 -8027.273,E2 -8027.273} C_VEL
LIN {X 0,Y 462.077,Z 326.49,A -85,B 0,C 180,E1 -8030.245,E2 -8030.245} C_VEL
LIN {X 0,Y 462.961,Z 308.249,A -85,B 0,C 180,E1 -8033.485,E2 -8033.485} C_VEL
LIN {X 0,Y 462.681,Z 303.831,A -85,B 0,C 180,E1 -8034.302,E2 -8034.302} C_VEL
LIN {X 0,Y 460.6,Z 293.113,A -85,B 0,C 180,E1 -8036.386,E2 -8036.386} C_VEL
LIN {X 0,Y 460.535,Z 293.12,A -85,B 0,C 180,E1 -8039.558,E2 -8039.558} C_VEL
LIN {X 0,Y 460.535,Z 293.12,A -85,B 0,C 180,E1 -8042.285,E2 -8042.285} C_VEL
LIN {X 0,Y 460.513,Z 293.117,A -85,B 0,C 180,E1 -8045.446,E2 -8045.446} C_VEL
LIN {X 0,Y 460.536,Z 293.115,A -85,B 0,C 180,E1 -8048.896,E2 -8048.896} C_VEL
LIN {X 0,Y 460.525,Z 293.121,A -85,B 0,C 180,E1 -8052.181,E2 -8052.181} C_VEL
LIN {X 0,Y 460.513,Z 293.116,A -85,B 0,C 180,E1 -8055.411,E2 -8055.411} C_VEL
LIN {X 0,Y 460.532,Z 293.121,A -85,B 0,C 180,E1 -8058.397,E2 -8058.397} C_VEL
LIN {X 0,Y 460.524,Z 293.116,A -85,B 0,C 180,E1 -8061.267,E2 -8061.267} C_VEL
LIN {X 0,Y 460.51,Z 293.124,A -85,B 0,C 180,E1 -8064.554,E2 -8064.554} C_VEL
LIN {X 0,Y 460.529,Z 293.114,A -85,B 0,C 180,E1 -8067.715,E2 -8067.715} C_VEL
LIN {X 0,Y 460.536,Z 293.122,A -85,B 0,C 180,E1 -8070.769,E2 -8070.769} C_VEL
LIN {X 0,Y 460.558,Z 293.111,A -85,B 0,C 180,E1 -8073.734,E2 -8073.734} C_VEL
LIN {X 0,Y 460.54,Z 293.117,A -85,B 0,C 180,E1 -8076.624,E2 -8076.624} C_VEL
LIN {X 0,Y 460.543,Z 293.115,A -85,B 0,C 180,E1 -8079.452,E2 -8079.452} C_VEL
LIN {X 0,Y 460.549,Z 293.112,A -85,B 0,C 180,E1 -8082.23,E2 -8082.23} C_VEL
LIN {X 0,Y 460.556,Z 293.117,A -85,B 0,C 180,E1 -8084.965,E2 -8084.965} C_VEL
LIN {X 0,Y 460.602,Z 293.106,A -85,B 0,C 180,E1 -8088.559,E2 -8088.559} C_VEL
LIN {X 0,Y 460.687,Z 293.095,A -85,B 0,C 180,E1 -8092.108,E2 -8092.108} C_VEL
LIN {X 0,Y 460.682,Z 293.096,A -85,B 0,C 180,E1 -8094.748,E2 -8094.748} C_VEL
LIN {X 0,Y 460.788,Z 293.09,A -85,B 0,C 180,E1 -8097.377,E2 -8097.377} C_VEL
LIN {X 0,Y 460.837,Z 293.078,A -85,B 0,C 180,E1 -8100,E2 -8100} C_VEL
LIN {X 0,Y 460.787,Z 293.082,A -85,B 0,C 180,E1 -8102.623,E2 -8102.623} C_VEL
LIN {X 0,Y 460.672,Z 293.099,A -85,B 0,C 180,E1 -8106.13,E2 -8106.13} C_VEL
LIN {X 0,Y 460.61,Z 293.104,A -85,B 0,C 180,E1 -8108.777,E2 -8108.777} C_VEL
LIN {X 0,Y 460.6,Z 293.107,A -85,B 0,C 180,E1 -8112.334,E2 -8112.334} C_VEL
LIN {X 0,Y 460.594,Z 293.113,A -85,B 0,C 180,E1 -8115.998,E2 -8115.998} C_VEL
LIN {X 0,Y 460.558,Z 293.115,A -85,B 0,C 180,E1 -8119.616,E2 -8119.616} C_VEL
LIN {X 0,Y 460.499,Z 293.121,A -85,B 0,C 180,E1 -8122.429,E2 -8122.429} C_VEL
LIN {X 0,Y 460.526,Z 293.119,A -85,B 0,C 180,E1 -8125.793,E2 -8125.793} C_VEL
LIN {X 0,Y 460.513,Z 293.116,A -85,B 0,C 180,E1 -8129.233,E2 -8129.233} C_VEL
LIN {X 0,Y 460.514,Z 293.125,A -85,B 0,C 180,E1 -8132.286,E2 -8132.286} C_VEL
LIN {X 0,Y 460.495,Z 293.118,A -85,B 0,C 180,E1 -8135.447,E2 -8135.447} C_VEL
LIN {X 0,Y 460.479,Z 293.123,A -85,B 0,C 180,E1 -8138.888,E2 -8138.888} C_VEL
LIN {X 0,Y 460.493,Z 293.119,A -85,B 0,C 180,E1 -8141.597,E2 -8141.597} C_VEL
LIN {X 0,Y 460.504,Z 293.126,A -85,B 0,C 180,E1 -8144.59,E2 -8144.59} C_VEL
LIN {X 0,Y 460.471,Z 293.122,A -85,B 0,C 180,E1 -8147.813,E2 -8147.813} C_VEL
LIN {X 0,Y 460.474,Z 293.123,A -85,B 0,C 180,E1 -8150.131,E2 -8150.131} C_VEL
LIN {X 0,Y 460.472,Z 293.127,A -85,B 0,C 180,E1 -8152.529,E2 -8152.529} C_VEL
LIN {X 0,Y 460.46,Z 293.123,A -85,B 0,C 180,E1 -8155.616,E2 -8155.616} C_VEL
LIN {X 0,Y 460.508,Z 293.123,A -85,B 0,C 180,E1 -8158.741,E2 -8158.741} C_VEL
LIN {X 0,Y 460.499,Z 293.118,A -85,B 0,C 180,E1 -8161.762,E2 -8161.762} C_VEL
LIN {X 0,Y 460.511,Z 293.121,A -85,B 0,C 180,E1 -8164.701,E2 -8164.701} C_VEL
LIN {X 0,Y 460.512,Z 293.119,A -85,B 0,C 180,E1 -8167.57,E2 -8167.57} C_VEL
LIN {X 0,Y 460.57,Z 293.11,A -85,B 0,C 180,E1 -8170.383,E2 -8170.383} C_VEL
LIN {X 0,Y 460.592,Z 293.107,A -85,B 0,C 180,E1 -8174.057,E2 -8174.057} C_VEL
LIN {X 0,Y 460.615,Z 293.108,A -85,B 0,C 180,E1 -8177.664,E2 -8177.664} C_VEL
LIN {X 0,Y 460.57,Z 293.114,A -85,B 0,C 180,E1 -8179.208,E2 -8179.208} C_VEL
LIN {X 0,Y 459.904,Z 293.202,A -85,B 0,C 180,E1 -8179.937,E2 -8179.937} C_VEL
LIN {X 0,Y 457.066,Z 293.556,A -85,B 0,C 180,E1 -8181.123,E2 -8181.123} C_VEL
LIN {X 0,Y 454.677,Z 293.848,A -85,B 0,C 180,E1 -8182.079,E2 -8182.079} C_VEL
LIN {X 0,Y 453.665,Z 293.971,A -85,B 0,C 180,E1 -8182.818,E2 -8182.818} C_VEL
LIN {X 0,Y 453.589,Z 293.98,A -85,B 0,C 180,E1 -8183.068,E2 -8183.068} C_VEL
LIN {X 0,Y 453.652,Z 293.971,A -85,B 0,C 180,E1 -8184.664,E2 -8184.664} C_VEL
LIN {X 0,Y 453.689,Z 293.967,A -85,B 0,C 180,E1 -8188.222,E2 -8188.222} C_VEL
LIN {X 0,Y 453.791,Z 293.957,A -85,B 0,C 180,E1 -8189.997,E2 -8189.997} C_VEL
LIN {X 0,Y 453.707,Z 293.964,A -85,B 0,C 180,E1 -8192.66,E2 -8192.66} C_VEL
LIN {X 0,Y 453.637,Z 293.978,A -85,B 0,C 180,E1 -8196.223,E2 -8196.223} C_VEL
LIN {X 0,Y 453.581,Z 293.984,A -85,B 0,C 180,E1 -8198.91,E2 -8198.91} C_VEL
LIN {X 0,Y 453.575,Z 294.105,A -85,B 0,C 180,E1 -8200.769,E2 -8200.769} C_VEL
LIN {X 0,Y 454.79,Z 301.811,A -85,B 0,C 180,E1 -8202.491,E2 -8202.491} C_VEL
LIN {X 0,Y 454.578,Z 311.667,A -85,B 0,C 180,E1 -8204.546,E2 -8204.546} C_VEL
LIN {X 0,Y 457.698,Z 327.43,A -85,B 0,C 180,E1 -8204.928,E2 -8204.928} C_VEL
LIN {X 0,Y 456.784,Z 418.996,A -85,B 0,C 180,E1 -8206.418,E2 -8206.418} C_VEL
LIN {X 0,Y 456.525,Z 432.594,A -85,B 0,C 180,E1 -8206.83,E2 -8206.83} C_VEL
LIN {X 0,Y 456.172,Z 444.76,A -85,B 0,C 180,E1 -8207.374,E2 -8207.374} C_VEL
LIN {X 0,Y 455.671,Z 456.458,A -85,B 0,C 180,E1 -8208.079,E2 -8208.079} C_VEL
LIN {X 0,Y 455.139,Z 467.323,A -85,B 0,C 180,E1 -8208.917,E2 -8208.917} C_VEL
LIN {X 0,Y 454.541,Z 478.521,A -85,B 0,C 180,E1 -8210,E2 -8210} C_VEL
LIN {X 0,Y 454.033,Z 487.532,A -85,B 0,C 180,E1 -8211.086,E2 -8211.086} C_VEL
LIN {X 0,Y 453.66,Z 495.744,A -85,B 0,C 180,E1 -8212.301,E2 -8212.301} C_VEL
LIN {X 0,Y 453.22,Z 503.95,A -85,B 0,C 180,E1 -8213.808,E2 -8213.808} C_VEL
LIN {X 0,Y 452.923,Z 510.079,A -85,B 0,C 180,E1 -8215.254,E2 -8215.254} C_VEL
LIN {X 0,Y 452.714,Z 514.946,A -85,B 0,C 180,E1 -8216.751,E2 -8216.751} C_VEL
LIN {X 0,Y 452.587,Z 517.504,A -85,B 0,C 180,E1 -8217.76,E2 -8217.76} C_VEL
LIN {X 0,Y 452.416,Z 520.596,A -85,B 0,C 180,E1 -8219.55,E2 -8219.55} C_VEL
LIN {X 0,Y 452.38,Z 522.069,A -85,B 0,C 180,E1 -8221.3,E2 -8221.3} C_VEL
LIN {X 0,Y 452.339,Z 522.008,A -85,B 0,C 180,E1 -8222.965,E2 -8222.965} C_VEL
LIN {X 0,Y 452.395,Z 520.635,A -85,B 0,C 180,E1 -8224.577,E2 -8224.577} C_VEL
LIN {X 0,Y 452.577,Z 518.005,A -85,B 0,C 180,E1 -8226.157,E2 -8226.157} C_VEL
LIN {X 0,Y 452.732,Z 514.261,A -85,B 0,C 180,E1 -8227.655,E2 -8227.655} C_VEL
LIN {X 0,Y 452.986,Z 509.225,A -85,B 0,C 180,E1 -8229.127,E2 -8229.127} C_VEL
LIN {X 0,Y 453.277,Z 502.58,A -85,B 0,C 180,E1 -8230.625,E2 -8230.625} C_VEL
LIN {X 0,Y 453.683,Z 495.108,A -85,B 0,C 180,E1 -8231.964,E2 -8231.964} C_VEL
LIN {X 0,Y 454.181,Z 487.027,A -85,B 0,C 180,E1 -8233.136,E2 -8233.136} C_VEL
LIN {X 0,Y 454.704,Z 477.732,A -85,B 0,C 180,E1 -8234.235,E2 -8234.235} C_VEL
LIN {X 0,Y 455.242,Z 467.283,A -85,B 0,C 180,E1 -8235.239,E2 -8235.239} C_VEL
LIN {X 0,Y 455.789,Z 456.587,A -85,B 0,C 180,E1 -8236.062,E2 -8236.062} C_VEL
LIN {X 0,Y 456.257,Z 444.732,A -85,B 0,C 180,E1 -8236.776,E2 -8236.776} C_VEL
LIN {X 0,Y 456.694,Z 431.207,A -85,B 0,C 180,E1 -8237.366,E2 -8237.366} C_VEL
LIN {X 0,Y 456.973,Z 418.53,A -85,B 0,C 180,E1 -8237.734,E2 -8237.734} C_VEL
LIN {X 0,Y 457.85,Z 327.353,A -85,B 0,C 180,E1 -8239.222,E2 -8239.222} C_VEL
LIN {X 0,Y 454.624,Z 311.134,A -85,B 0,C 180,E1 -8239.64,E2 -8239.64} C_VEL
LIN {X 0,Y 454.76,Z 301.072,A -85,B 0,C 180,E1 -8241.535,E2 -8241.535} C_VEL
LIN {X 0,Y 453.461,Z 294.001,A -85,B 0,C 180,E1 -8242.963,E2 -8242.963} C_VEL
LIN {X 0,Y 453.438,Z 294.006,A -85,B 0,C 180,E1 -8246.084,E2 -8246.084} C_VEL
LIN {X 0,Y 453.441,Z 294.001,A -85,B 0,C 180,E1 -8249.238,E2 -8249.238} C_VEL
LIN {X 0,Y 453.5,Z 294.002,A -85,B 0,C 180,E1 -8252.295,E2 -8252.295} C_VEL
LIN {X 0,Y 453.468,Z 294,A -85,B 0,C 180,E1 -8255.263,E2 -8255.263} C_VEL
LIN {X 0,Y 453.432,Z 294.009,A -85,B 0,C 180,E1 -8258.413,E2 -8258.413} C_VEL
LIN {X 0,Y 453.473,Z 293.997,A -85,B 0,C 180,E1 -8261.006,E2 -8261.006} C_VEL
LIN {X 0,Y 453.519,Z 293.99,A -85,B 0,C 180,E1 -8263.878,E2 -8263.878} C_VEL
LIN {X 0,Y 453.512,Z 293.99,A -85,B 0,C 180,E1 -8267.47,E2 -8267.47} C_VEL
LIN {X 0,Y 453.54,Z 293.989,A -85,B 0,C 180,E1 -8271.086,E2 -8271.086} C_VEL
LIN {X 0,Y 453.618,Z 293.976,A -85,B 0,C 180,E1 -8273.774,E2 -8273.774} C_VEL
LIN {X 0,Y 453.718,Z 293.966,A -85,B 0,C 180,E1 -8277.337,E2 -8277.337} C_VEL
LIN {X 0,Y 453.767,Z 293.953,A -85,B 0,C 180,E1 -8280,E2 -8280} C_VEL
LIN {X 0,Y 453.72,Z 293.968,A -85,B 0,C 180,E1 -8282.663,E2 -8282.663} C_VEL
LIN {X 0,Y 453.629,Z 293.975,A -85,B 0,C 180,E1 -8286.226,E2 -8286.226} C_VEL
LIN {X 0,Y 453.546,Z 293.987,A -85,B 0,C 180,E1 -8288.914,E2 -8288.914} C_VEL
LIN {X 0,Y 453.551,Z 293.981,A -85,B 0,C 180,E1 -8292.552,E2 -8292.552} C_VEL
LIN {X 0,Y 453.506,Z 293.985,A -85,B 0,C 180,E1 -8296.197,E2 -8296.197} C_VEL
LIN {X 0,Y 453.472,Z 293.999,A -85,B 0,C 180,E1 -8299.043,E2 -8299.043} C_VEL
LIN {X 0,Y 453.458,Z 293.996,A -85,B 0,C 180,E1 -8301.837,E2 -8301.837} C_VEL
LIN {X 0,Y 453.487,Z 293.988,A -85,B 0,C 180,E1 -8304.736,E2 -8304.736} C_VEL
LIN {X 0,Y 453.495,Z 293.989,A -85,B 0,C 180,E1 -8307.964,E2 -8307.964} C_VEL
LIN {X 0,Y 453.441,Z 293.999,A -85,B 0,C 180,E1 -8310.762,E2 -8310.762} C_VEL
LIN {X 0,Y 453.439,Z 294.001,A -85,B 0,C 180,E1 -8313.916,E2 -8313.916} C_VEL
LIN {X 0,Y 453.442,Z 294.002,A -85,B 0,C 180,E1 -8317.191,E2 -8317.191} C_VEL
LIN {X 0,Y 453.51,Z 293.995,A -85,B 0,C 180,E1 -8319.448,E2 -8319.448} C_VEL
LIN {X 0,Y 453.459,Z 294,A -85,B 0,C 180,E1 -8322.996,E2 -8322.996} C_VEL
LIN {X 0,Y 453.447,Z 294.006,A -85,B 0,C 180,E1 -8325.785,E2 -8325.785} C_VEL
LIN {X 0,Y 453.469,Z 294,A -85,B 0,C 180,E1 -8328.216,E2 -8328.216} C_VEL
LIN {X 0,Y 453.51,Z 293.992,A -85,B 0,C 180,E1 -8330.791,E2 -8330.791} C_VEL
LIN {X 0,Y 453.435,Z 294.003,A -85,B 0,C 180,E1 -8333.922,E2 -8333.922} C_VEL
LIN {X 0,Y 453.464,Z 294.001,A -85,B 0,C 180,E1 -8337.156,E2 -8337.156} C_VEL
LIN {X 0,Y 453.497,Z 293.999,A -85,B 0,C 180,E1 -8340.276,E2 -8340.276} C_VEL
LIN {X 0,Y 453.548,Z 293.992,A -85,B 0,C 180,E1 -8343.637,E2 -8343.637} C_VEL
LIN {X 0,Y 455.814,Z 305.78,A -85,B 0,C 180,E1 -8345.94,E2 -8345.94} C_VEL
LIN {X 0,Y 455.334,Z 318.881,A -85,B 0,C 180,E1 -8348.262,E2 -8348.262} C_VEL
LIN {X 0,Y 454.557,Z 337.547,A -85,B 0,C 180,E1 -8351.526,E2 -8351.526} C_VEL
LIN {X 0,Y 454.353,Z 342.604,A -85,B 0,C 180,E1 -8352.402,E2 -8352.402} C_VEL
LIN {X 0,Y 457.638,Z 365.333,A -85,B 0,C 180,E1 -8352.913,E2 -8352.913} C_VEL
LIN {X 0,Y 456.783,Z 451.835,A -85,B 0,C 180,E1 -8354.327,E2 -8354.327} C_VEL
LIN {X 0,Y 456.349,Z 465.631,A -85,B 0,C 180,E1 -8354.741,E2 -8354.741} C_VEL
LIN {X 0,Y 455.775,Z 478.556,A -85,B 0,C 180,E1 -8355.321,E2 -8355.321} C_VEL
LIN {X 0,Y 455.276,Z 490.348,A -85,B 0,C 180,E1 -8356.047,E2 -8356.047} C_VEL
LIN {X 0,Y 454.751,Z 501.555,A -85,B 0,C 180,E1 -8356.925,E2 -8356.925} C_VEL
LIN {X 0,Y 454.208,Z 512.002,A -85,B 0,C 180,E1 -8357.947,E2 -8357.947} C_VEL
LIN {X 0,Y 453.645,Z 521.237,A -85,B 0,C 180,E1 -8359.064,E2 -8359.064} C_VEL
LIN {X 0,Y 453.195,Z 530.241,A -85,B 0,C 180,E1 -8360.407,E2 -8360.407} C_VEL
LIN {X 0,Y 452.901,Z 537.494,A -85,B 0,C 180,E1 -8361.751,E2 -8361.751} C_VEL
LIN {X 0,Y 452.714,Z 542.391,A -85,B 0,C 180,E1 -8362.869,E2 -8362.869} C_VEL
LIN {X 0,Y 452.556,Z 547.152,A -85,B 0,C 180,E1 -8364.21,E2 -8364.21} C_VEL
LIN {X 0,Y 452.485,Z 550.793,A -85,B 0,C 180,E1 -8365.549,E2 -8365.549} C_VEL
LIN {X 0,Y 452.482,Z 552.672,A -85,B 0,C 180,E1 -8366.441,E2 -8366.441} C_VEL
LIN {X 0,Y 452.507,Z 554.083,A -85,B 0,C 180,E1 -8367.332,E2 -8367.332} C_VEL
LIN {X 0,Y 452.457,Z 555.706,A -85,B 0,C 180,E1 -8369.113,E2 -8369.113} C_VEL
LIN {X 0,Y 452.465,Z 555.924,A -85,B 0,C 180,E1 -8370.003,E2 -8370.003} C_VEL
LIN {X 0,Y 452.457,Z 555.705,A -85,B 0,C 180,E1 -8370.893,E2 -8370.893} C_VEL
LIN {X 0,Y 452.508,Z 554.093,A -85,B 0,C 180,E1 -8372.673,E2 -8372.673} C_VEL
LIN {X 0,Y 452.483,Z 552.678,A -85,B 0,C 180,E1 -8373.565,E2 -8373.565} C_VEL
LIN {X 0,Y 452.546,Z 549.717,A -85,B 0,C 180,E1 -8374.902,E2 -8374.902} C_VEL
LIN {X 0,Y 452.613,Z 545.15,A -85,B 0,C 180,E1 -8376.398,E2 -8376.398} C_VEL
LIN {X 0,Y 452.846,Z 538.503,A -85,B 0,C 180,E1 -8378.031,E2 -8378.031} C_VEL
LIN {X 0,Y 453.122,Z 531.525,A -85,B 0,C 180,E1 -8379.375,E2 -8379.375} C_VEL
LIN {X 0,Y 453.543,Z 522.775,A -85,B 0,C 180,E1 -8380.719,E2 -8380.719} C_VEL
LIN {X 0,Y 454.095,Z 513.819,A -85,B 0,C 180,E1 -8381.836,E2 -8381.836} C_VEL
LIN {X 0,Y 454.519,Z 504.703,A -85,B 0,C 180,E1 -8382.774,E2 -8382.774} C_VEL
LIN {X 0,Y 455.113,Z 493.142,A -85,B 0,C 180,E1 -8383.737,E2 -8383.737} C_VEL
LIN {X 0,Y 455.681,Z 480.988,A -85,B 0,C 180,E1 -8384.516,E2 -8384.516} C_VEL
LIN {X 0,Y 456.191,Z 468.3,A -85,B 0,C 180,E1 -8385.127,E2 -8385.127} C_VEL
LIN {X 0,Y 456.584,Z 455.825,A -85,B 0,C 180,E1 -8385.543,E2 -8385.543} C_VEL
LIN {X 0,Y 456.913,Z 440.075,A -85,B 0,C 180,E1 -8385.846,E2 -8385.846} C_VEL
LIN {X 0,Y 457.425,Z 363.324,A -85,B 0,C 180,E1 -8387.082,E2 -8387.082} C_VEL
LIN {X 0,Y 454.332,Z 343.244,A -85,B 0,C 180,E1 -8387.535,E2 -8387.535} C_VEL
LIN {X 0,Y 455.102,Z 327.511,A -85,B 0,C 180,E1 -8390.334,E2 -8390.334} C_VEL
LIN {X 0,Y 456.036,Z 309.265,A -85,B 0,C 180,E1 -8393.623,E2 -8393.623} C_VEL
LIN {X 0,Y 455.641,Z 304.692,A -85,B 0,C 180,E1 -8394.489,E2 -8394.489} C_VEL
LIN {X 0,Y 453.577,Z 293.988,A -85,B 0,C 180,E1 -8396.617,E2 -8396.617} C_VEL
LIN {X 0,Y 453.476,Z 294,A -85,B 0,C 180,E1 -8399.785,E2 -8399.785} C_VEL
LIN {X 0,Y 453.493,Z 293.991,A -85,B 0,C 180,E1 -8403.189,E2 -8403.189} C_VEL
LIN {X 0,Y 453.456,Z 294.003,A -85,B 0,C 180,E1 -8406.299,E2 -8406.299} C_VEL
LIN {X 0,Y 453.47,Z 293.994,A -85,B 0,C 180,E1 -8409.452,E2 -8409.452} C_VEL
LIN {X 0,Y 453.478,Z 293.996,A -85,B 0,C 180,E1 -8411.935,E2 -8411.935} C_VEL
LIN {X 0,Y 453.483,Z 293.992,A -85,B 0,C 180,E1 -8415.471,E2 -8415.471} C_VEL
LIN {X 0,Y 453.479,Z 293.997,A -85,B 0,C 180,E1 -8418.209,E2 -8418.209} C_VEL
LIN {X 0,Y 453.509,Z 293.994,A -85,B 0,C 180,E1 -8420.791,E2 -8420.791} C_VEL
LIN {X 0,Y 453.453,Z 293.996,A -85,B 0,C 180,E1 -8423.917,E2 -8423.917} C_VEL
LIN {X 0,Y 453.48,Z 293.995,A -85,B 0,C 180,E1 -8427.151,E2 -8427.151} C_VEL
LIN {X 0,Y 453.472,Z 293.996,A -85,B 0,C 180,E1 -8430.268,E2 -8430.268} C_VEL
LIN {X 0,Y 453.502,Z 293.992,A -85,B 0,C 180,E1 -8433.294,E2 -8433.294} C_VEL
LIN {X 0,Y 453.497,Z 293.991,A -85,B 0,C 180,E1 -8436.238,E2 -8436.238} C_VEL
LIN {X 0,Y 453.476,Z 294,A -85,B 0,C 180,E1 -8439.117,E2 -8439.117} C_VEL
LIN {X 0,Y 453.502,Z 293.99,A -85,B 0,C 180,E1 -8441.944,E2 -8441.944} C_VEL
LIN {X 0,Y 453.531,Z 293.989,A -85,B 0,C 180,E1 -8444.726,E2 -8444.726} C_VEL
LIN {X 0,Y 453.551,Z 293.984,A -85,B 0,C 180,E1 -8448.379,E2 -8448.379} C_VEL
LIN {X 0,Y 453.644,Z 293.973,A -85,B 0,C 180,E1 -8451.985,E2 -8451.985} C_VEL
LIN {X 0,Y 453.656,Z 293.971,A -85,B 0,C 180,E1 -8454.667,E2 -8454.667} C_VEL
LIN {X 0,Y 453.732,Z 293.968,A -85,B 0,C 180,E1 -8457.337,E2 -8457.337} C_VEL
LIN {X 0,Y 453.808,Z 293.954,A -85,B 0,C 180,E1 -8460,E2 -8460} C_VEL
LIN {X 0,Y 453.732,Z 293.961,A -85,B 0,C 180,E1 -8462.663,E2 -8462.663} C_VEL
LIN {X 0,Y 453.639,Z 293.974,A -85,B 0,C 180,E1 -8466.226,E2 -8466.226} C_VEL
LIN {X 0,Y 453.576,Z 293.981,A -85,B 0,C 180,E1 -8468.914,E2 -8468.914} C_VEL
LIN {X 0,Y 453.557,Z 293.983,A -85,B 0,C 180,E1 -8472.529,E2 -8472.529} C_VEL
LIN {X 0,Y 453.538,Z 293.989,A -85,B 0,C 180,E1 -8476.196,E2 -8476.196} C_VEL
LIN {X 0,Y 453.511,Z 293.989,A -85,B 0,C 180,E1 -8479.039,E2 -8479.039} C_VEL
LIN {X 0,Y 453.469,Z 294,A -85,B 0,C 180,E1 -8481.837,E2 -8481.837} C_VEL
LIN {X 0,Y 453.461,Z 293.996,A -85,B 0,C 180,E1 -8484.738,E2 -8484.738} C_VEL
LIN {X 0,Y 453.455,Z 294.001,A -85,B 0,C 180,E1 -8487.942,E2 -8487.942} C_VEL
LIN {X 0,Y 453.453,Z 293.998,A -85,B 0,C 180,E1 -8490.761,E2 -8490.761} C_VEL
LIN {X 0,Y 453.461,Z 293.998,A -85,B 0,C 180,E1 -8493.914,E2 -8493.914} C_VEL
LIN {X 0,Y 453.431,Z 293.999,A -85,B 0,C 180,E1 -8497.192,E2 -8497.192} C_VEL
LIN {X 0,Y 453.465,Z 294.001,A -85,B 0,C 180,E1 -8500.612,E2 -8500.612} C_VEL
LIN {X 0,Y 453.476,Z 294.001,A -85,B 0,C 180,E1 -8504.528,E2 -8504.528} C_VEL
LIN {X 0,Y 453.437,Z 294.001,A -85,B 0,C 180,E1 -8508.204,E2 -8508.204} C_VEL
LIN {X 0,Y 453.422,Z 294.007,A -85,B 0,C 180,E1 -8510.805,E2 -8510.805} C_VEL
LIN {X 0,Y 453.402,Z 294.002,A -85,B 0,C 180,E1 -8513.912,E2 -8513.912} C_VEL
LIN {X 0,Y 453.436,Z 294.002,A -85,B 0,C 180,E1 -8517.146,E2 -8517.146} C_VEL
LIN {X 0,Y 453.451,Z 293.997,A -85,B 0,C 180,E1 -8520.266,E2 -8520.266} C_VEL
LIN {X 0,Y 453.423,Z 294.004,A -85,B 0,C 180,E1 -8523.287,E2 -8523.287} C_VEL
LIN {X 0,Y 453.495,Z 293.991,A -85,B 0,C 180,E1 -8526.237,E2 -8526.237} C_VEL
LIN {X 0,Y 453.487,Z 294,A -85,B 0,C 180,E1 -8529.116,E2 -8529.116} C_VEL
LIN {X 0,Y 453.5,Z 293.99,A -85,B 0,C 180,E1 -8531.942,E2 -8531.942} C_VEL
LIN {X 0,Y 453.536,Z 293.987,A -85,B 0,C 180,E1 -8534.724,E2 -8534.724} C_VEL
LIN {X 0,Y 453.562,Z 293.982,A -85,B 0,C 180,E1 -8538.377,E2 -8538.377} C_VEL
LIN {X 0,Y 453.565,Z 293.986,A -85,B 0,C 180,E1 -8541.084,E2 -8541.084} C_VEL
LIN {X 0,Y 453.589,Z 293.98,A -85,B 0,C 180,E1 -8543.068,E2 -8543.068} C_VEL
LIN {X 0,Y 452.909,Z 294.068,A -85,B 0,C 180,E1 -8543.809,E2 -8543.809} C_VEL
LIN {X 0,Y 449.96,Z 294.433,A -85,B 0,C 180,E1 -8545.011,E2 -8545.011} C_VEL
LIN {X 0,Y 447.53,Z 294.736,A -85,B 0,C 180,E1 -8545.981,E2 -8545.981} C_VEL
LIN {X 0,Y 446.588,Z 294.852,A -85,B 0,C 180,E1 -8546.731,E2 -8546.731} C_VEL
LIN {X 0,Y 446.566,Z 294.855,A -85,B 0,C 180,E1 -8546.985,E2 -8546.985} C_VEL
LIN {X 0,Y 446.74,Z 294.836,A -85,B 0,C 180,E1 -8549.997,E2 -8549.997} C_VEL
LIN {X 0,Y 446.657,Z 294.842,A -85,B 0,C 180,E1 -8552.702,E2 -8552.702} C_VEL
LIN {X 0,Y 446.606,Z 294.854,A -85,B 0,C 180,E1 -8556.321,E2 -8556.321} C_VEL
LIN {X 0,Y 446.529,Z 294.863,A -85,B 0,C 180,E1 -8559.052,E2 -8559.052} C_VEL
LIN {X 0,Y 446.549,Z 295.056,A -85,B 0,C 180,E1 -8560.596,E2 -8560.596} C_VEL
LIN {X 0,Y 447.843,Z 303.273,A -85,B 0,C 180,E1 -8562.457,E2 -8562.457} C_VEL
LIN {X 0,Y 447.611,Z 311.669,A -85,B 0,C 180,E1 -8564.255,E2 -8564.255} C_VEL
LIN {X 0,Y 450.938,Z 328.705,A -85,B 0,C 180,E1 -8564.689,E2 -8564.689} C_VEL
LIN {X 0,Y 449.967,Z 419.001,A -85,B 0,C 180,E1 -8566.178,E2 -8566.178} C_VEL
LIN {X 0,Y 449.692,Z 432.686,A -85,B 0,C 180,E1 -8566.597,E2 -8566.597} C_VEL
LIN {X 0,Y 449.324,Z 444.108,A -85,B 0,C 180,E1 -8567.108,E2 -8567.108} C_VEL
LIN {X 0,Y 448.853,Z 455.327,A -85,B 0,C 180,E1 -8567.773,E2 -8567.773} C_VEL
LIN {X 0,Y 448.306,Z 466.465,A -85,B 0,C 180,E1 -8568.623,E2 -8568.623} C_VEL
LIN {X 0,Y 447.676,Z 476.917,A -85,B 0,C 180,E1 -8569.621,E2 -8569.621} C_VEL
LIN {X 0,Y 447.183,Z 486.121,A -85,B 0,C 180,E1 -8570.704,E2 -8570.704} C_VEL
LIN {X 0,Y 446.716,Z 494.737,A -85,B 0,C 180,E1 -8571.944,E2 -8571.944} C_VEL
LIN {X 0,Y 446.307,Z 501.72,A -85,B 0,C 180,E1 -8573.178,E2 -8573.178} C_VEL
LIN {X 0,Y 445.946,Z 508.509,A -85,B 0,C 180,E1 -8574.68,E2 -8574.68} C_VEL
LIN {X 0,Y 445.721,Z 513.823,A -85,B 0,C 180,E1 -8576.194,E2 -8576.194} C_VEL
LIN {X 0,Y 445.476,Z 518.249,A -85,B 0,C 180,E1 -8577.935,E2 -8577.935} C_VEL
LIN {X 0,Y 445.311,Z 521.176,A -85,B 0,C 180,E1 -8579.77,E2 -8579.77} C_VEL
LIN {X 0,Y 445.277,Z 522.393,A -85,B 0,C 180,E1 -8581.536,E2 -8581.536} C_VEL
LIN {X 0,Y 445.266,Z 522.15,A -85,B 0,C 180,E1 -8583.223,E2 -8583.223} C_VEL
LIN {X 0,Y 445.348,Z 520.617,A -85,B 0,C 180,E1 -8584.854,E2 -8584.854} C_VEL
LIN {X 0,Y 445.55,Z 517.831,A -85,B 0,C 180,E1 -8586.441,E2 -8586.441} C_VEL
LIN {X 0,Y 445.71,Z 513.872,A -85,B 0,C 180,E1 -8587.963,E2 -8587.963} C_VEL
LIN {X 0,Y 445.971,Z 508.681,A -85,B 0,C 180,E1 -8589.449,E2 -8589.449} C_VEL
LIN {X 0,Y 446.292,Z 502.205,A -85,B 0,C 180,E1 -8590.897,E2 -8590.897} C_VEL
LIN {X 0,Y 446.762,Z 494.13,A -85,B 0,C 180,E1 -8592.323,E2 -8592.323} C_VEL
LIN {X 0,Y 447.344,Z 485.338,A -85,B 0,C 180,E1 -8593.567,E2 -8593.567} C_VEL
LIN {X 0,Y 447.986,Z 475.098,A -85,B 0,C 180,E1 -8594.74,E2 -8594.74} C_VEL
LIN {X 0,Y 448.488,Z 464.766,A -85,B 0,C 180,E1 -8595.69,E2 -8595.69} C_VEL
LIN {X 0,Y 449.073,Z 453.969,A -85,B 0,C 180,E1 -8596.48,E2 -8596.48} C_VEL
LIN {X 0,Y 449.556,Z 442.113,A -85,B 0,C 180,E1 -8597.157,E2 -8597.157} C_VEL
LIN {X 0,Y 449.957,Z 429.233,A -85,B 0,C 180,E1 -8597.692,E2 -8597.692} C_VEL
LIN {X 0,Y 450.218,Z 415.724,A -85,B 0,C 180,E1 -8598.045,E2 -8598.045} C_VEL
LIN {X 0,Y 451.065,Z 327.867,A -85,B 0,C 180,E1 -8599.494,E2 -8599.494} C_VEL
LIN {X 0,Y 447.685,Z 311.362,A -85,B 0,C 180,E1 -8599.936,E2 -8599.936} C_VEL
LIN {X 0,Y 447.76,Z 301.501,A -85,B 0,C 180,E1 -8601.823,E2 -8601.823} C_VEL
LIN {X 0,Y 446.422,Z 294.877,A -85,B 0,C 180,E1 -8603.186,E2 -8603.186} C_VEL
LIN {X 0,Y 446.409,Z 294.881,A -85,B 0,C 180,E1 -8606.563,E2 -8606.563} C_VEL
LIN {X 0,Y 446.398,Z 294.882,A -85,B 0,C 180,E1 -8609.974,E2 -8609.974} C_VEL
LIN {X 0,Y 446.437,Z 294.878,A -85,B 0,C 180,E1 -8612.836,E2 -8612.836} C_VEL
LIN {X 0,Y 446.419,Z 294.881,A -85,B 0,C 180,E1 -8615.921,E2 -8615.921} C_VEL
LIN {X 0,Y 446.404,Z 294.882,A -85,B 0,C 180,E1 -8618.771,E2 -8618.771} C_VEL
LIN {X 0,Y 446.406,Z 294.876,A -85,B 0,C 180,E1 -8621.647,E2 -8621.647} C_VEL
LIN {X 0,Y 446.456,Z 294.874,A -85,B 0,C 180,E1 -8624.478,E2 -8624.478} C_VEL
LIN {X 0,Y 446.467,Z 294.87,A -85,B 0,C 180,E1 -8628.192,E2 -8628.192} C_VEL
LIN {X 0,Y 446.548,Z 294.857,A -85,B 0,C 180,E1 -8631.857,E2 -8631.857} C_VEL
LIN {X 0,Y 446.59,Z 294.857,A -85,B 0,C 180,E1 -8634.582,E2 -8634.582} C_VEL
LIN {X 0,Y 446.662,Z 294.845,A -85,B 0,C 180,E1 -8637.294,E2 -8637.294} C_VEL
LIN {X 0,Y 446.738,Z 294.828,A -85,B 0,C 180,E1 -8640,E2 -8640} C_VEL
LIN {X 0,Y 446.664,Z 294.848,A -85,B 0,C 180,E1 -8642.706,E2 -8642.706} C_VEL
LIN {X 0,Y 446.597,Z 294.852,A -85,B 0,C 180,E1 -8646.324,E2 -8646.324} C_VEL
LIN {X 0,Y 446.493,Z 294.868,A -85,B 0,C 180,E1 -8649.056,E2 -8649.056} C_VEL
LIN {X 0,Y 446.484,Z 294.863,A -85,B 0,C 180,E1 -8652.731,E2 -8652.731} C_VEL
LIN {X 0,Y 446.446,Z 294.865,A -85,B 0,C 180,E1 -8656.461,E2 -8656.461} C_VEL
LIN {X 0,Y 446.422,Z 294.875,A -85,B 0,C 180,E1 -8659.305,E2 -8659.305} C_VEL
LIN {X 0,Y 446.397,Z 294.874,A -85,B 0,C 180,E1 -8662.201,E2 -8662.201} C_VEL
LIN {X 0,Y 446.431,Z 294.871,A -85,B 0,C 180,E1 -8665.154,E2 -8665.154} C_VEL
LIN {X 0,Y 446.441,Z 294.866,A -85,B 0,C 180,E1 -8668.182,E2 -8668.182} C_VEL
LIN {X 0,Y 446.379,Z 294.882,A -85,B 0,C 180,E1 -8671.303,E2 -8671.303} C_VEL
LIN {X 0,Y 446.392,Z 294.876,A -85,B 0,C 180,E1 -8674.526,E2 -8674.526} C_VEL
LIN {X 0,Y 446.417,Z 294.875,A -85,B 0,C 180,E1 -8678.089,E2 -8678.089} C_VEL
LIN {X 0,Y 446.414,Z 294.875,A -85,B 0,C 180,E1 -8680.925,E2 -8680.925} C_VEL
LIN {X 0,Y 446.414,Z 294.882,A -85,B 0,C 180,E1 -8683.845,E2 -8683.845} C_VEL
LIN {X 0,Y 446.417,Z 294.878,A -85,B 0,C 180,E1 -8686.401,E2 -8686.401} C_VEL
LIN {X 0,Y 446.444,Z 294.878,A -85,B 0,C 180,E1 -8689.809,E2 -8689.809} C_VEL
LIN {X 0,Y 446.412,Z 294.88,A -85,B 0,C 180,E1 -8692.128,E2 -8692.128} C_VEL
LIN {X 0,Y 446.41,Z 294.88,A -85,B 0,C 180,E1 -8695.482,E2 -8695.482} C_VEL
LIN {X 0,Y 446.402,Z 294.882,A -85,B 0,C 180,E1 -8698.704,E2 -8698.704} C_VEL
LIN {X 0,Y 446.469,Z 294.874,A -85,B 0,C 180,E1 -8701.826,E2 -8701.826} C_VEL
LIN {X 0,Y 446.521,Z 295.052,A -85,B 0,C 180,E1 -8703.478,E2 -8703.478} C_VEL
LIN {X 0,Y 448.77,Z 306.3,A -85,B 0,C 180,E1 -8705.679,E2 -8705.679} C_VEL
LIN {X 0,Y 448.855,Z 310.618,A -85,B 0,C 180,E1 -8706.472,E2 -8706.472} C_VEL
LIN {X 0,Y 448.062,Z 326.654,A -85,B 0,C 180,E1 -8709.339,E2 -8709.339} C_VEL
LIN {X 0,Y 447.403,Z 342.301,A -85,B 0,C 180,E1 -8712.106,E2 -8712.106} C_VEL
LIN {X 0,Y 450.842,Z 365.295,A -85,B 0,C 180,E1 -8712.642,E2 -8712.642} C_VEL
LIN {X 0,Y 449.983,Z 450.698,A -85,B 0,C 180,E1 -8714.055,E2 -8714.055} C_VEL
LIN {X 0,Y 449.575,Z 464.006,A -85,B 0,C 180,E1 -8714.447,E2 -8714.447} C_VEL
LIN {X 0,Y 449.035,Z 476.211,A -85,B 0,C 180,E1 -8714.98,E2 -8714.98} C_VEL
LIN {X 0,Y 448.441,Z 488.552,A -85,B 0,C 180,E1 -8715.714,E2 -8715.714} C_VEL
LIN {X 0,Y 447.933,Z 499.16,A -85,B 0,C 180,E1 -8716.53,E2 -8716.53} C_VEL
LIN {X 0,Y 447.283,Z 510.699,A -85,B 0,C 180,E1 -8717.642,E2 -8717.642} C_VEL
LIN {X 0,Y 446.781,Z 519.291,A -85,B 0,C 180,E1 -8718.664,E2 -8718.664} C_VEL
LIN {X 0,Y 446.288,Z 527.226,A -85,B 0,C 180,E1 -8719.799,E2 -8719.799} C_VEL
LIN {X 0,Y 445.943,Z 534.982,A -85,B 0,C 180,E1 -8721.165,E2 -8721.165} C_VEL
LIN {X 0,Y 445.63,Z 542.134,A -85,B 0,C 180,E1 -8722.755,E2 -8722.755} C_VEL
LIN {X 0,Y 445.48,Z 546.337,A -85,B 0,C 180,E1 -8723.942,E2 -8723.942} C_VEL
LIN {X 0,Y 445.411,Z 550.536,A -85,B 0,C 180,E1 -8725.478,E2 -8725.478} C_VEL
LIN {X 0,Y 445.38,Z 552.413,A -85,B 0,C 180,E1 -8726.384,E2 -8726.384} C_VEL
LIN {X 0,Y 445.432,Z 553.823,A -85,B 0,C 180,E1 -8727.29,E2 -8727.29} C_VEL
LIN {X 0,Y 445.365,Z 555.444,A -85,B 0,C 180,E1 -8729.099,E2 -8729.099} C_VEL
LIN {X 0,Y 445.372,Z 555.659,A -85,B 0,C 180,E1 -8730.003,E2 -8730.003} C_VEL
LIN {X 0,Y 445.366,Z 555.437,A -85,B 0,C 180,E1 -8730.907,E2 -8730.907} C_VEL
LIN {X 0,Y 445.433,Z 553.822,A -85,B 0,C 180,E1 -8732.716,E2 -8732.716} C_VEL
LIN {X 0,Y 445.382,Z 552.402,A -85,B 0,C 180,E1 -8733.622,E2 -8733.622} C_VEL
LIN {X 0,Y 445.475,Z 549.437,A -85,B 0,C 180,E1 -8734.98,E2 -8734.98} C_VEL
LIN {X 0,Y 445.558,Z 543.961,A -85,B 0,C 180,E1 -8736.751,E2 -8736.751} C_VEL
LIN {X 0,Y 445.776,Z 538.203,A -85,B 0,C 180,E1 -8738.16,E2 -8738.16} C_VEL
LIN {X 0,Y 446.069,Z 531.214,A -85,B 0,C 180,E1 -8739.525,E2 -8739.525} C_VEL
LIN {X 0,Y 446.537,Z 522.451,A -85,B 0,C 180,E1 -8740.889,E2 -8740.889} C_VEL
LIN {X 0,Y 447.116,Z 513.48,A -85,B 0,C 180,E1 -8742.023,E2 -8742.023} C_VEL
LIN {X 0,Y 447.624,Z 503.337,A -85,B 0,C 180,E1 -8743.073,E2 -8743.073} C_VEL
LIN {X 0,Y 448.175,Z 492.753,A -85,B 0,C 180,E1 -8743.954,E2 -8743.954} C_VEL
LIN {X 0,Y 448.797,Z 480.567,A -85,B 0,C 180,E1 -8744.744,E2 -8744.744} C_VEL
LIN {X 0,Y 449.328,Z 467.83,A -85,B 0,C 180,E1 -8745.364,E2 -8745.364} C_VEL
LIN {X 0,Y 449.751,Z 455.203,A -85,B 0,C 180,E1 -8745.785,E2 -8745.785} C_VEL
LIN {X 0,Y 450.075,Z 437.499,A -85,B 0,C 180,E1 -8746.122,E2 -8746.122} C_VEL
LIN {X 0,Y 450.616,Z 364.172,A -85,B 0,C 180,E1 -8747.322,E2 -8747.322} C_VEL
LIN {X 0,Y 447.366,Z 342.991,A -85,B 0,C 180,E1 -8747.809,E2 -8747.809} C_VEL
LIN {X 0,Y 448.155,Z 327.209,A -85,B 0,C 180,E1 -8750.663,E2 -8750.663} C_VEL
LIN {X 0,Y 449.102,Z 310.286,A -85,B 0,C 180,E1 -8753.765,E2 -8753.765} C_VEL
LIN {X 0,Y 448.618,Z 305.525,A -85,B 0,C 180,E1 -8754.684,E2 -8754.684} C_VEL
LIN {X 0,Y 446.525,Z 294.866,A -85,B 0,C 180,E1 -8756.864,E2 -8756.864} C_VEL
LIN {X 0,Y 446.432,Z 294.879,A -85,B 0,C 180,E1 -8760.25,E2 -8760.25} C_VEL
LIN {X 0,Y 446.45,Z 294.869,A -85,B 0,C 180,E1 -8763.454,E2 -8763.454} C_VEL
LIN {X 0,Y 446.405,Z 294.876,A -85,B 0,C 180,E1 -8766.746,E2 -8766.746} C_VEL
LIN {X 0,Y 446.439,Z 294.877,A -85,B 0,C 180,E1 -8770.199,E2 -8770.199} C_VEL
LIN {X 0,Y 446.43,Z 294.876,A -85,B 0,C 180,E1 -8772.605,E2 -8772.605} C_VEL
LIN {X 0,Y 446.451,Z 294.869,A -85,B 0,C 180,E1 -8775.104,E2 -8775.104} C_VEL
LIN {X 0,Y 446.428,Z 294.878,A -85,B 0,C 180,E1 -8778.609,E2 -8778.609} C_VEL
LIN {X 0,Y 446.454,Z 294.871,A -85,B 0,C 180,E1 -8780.974,E2 -8780.974} C_VEL
LIN {X 0,Y 446.418,Z 294.877,A -85,B 0,C 180,E1 -8784.374,E2 -8784.374} C_VEL
LIN {X 0,Y 446.419,Z 294.872,A -85,B 0,C 180,E1 -8787.638,E2 -8787.638} C_VEL
LIN {X 0,Y 446.445,Z 294.878,A -85,B 0,C 180,E1 -8790.79,E2 -8790.79} C_VEL
LIN {X 0,Y 446.474,Z 294.865,A -85,B 0,C 180,E1 -8793.848,E2 -8793.848} C_VEL
LIN {X 0,Y 446.423,Z 294.878,A -85,B 0,C 180,E1 -8796.823,E2 -8796.823} C_VEL
LIN {X 0,Y 446.437,Z 294.87,A -85,B 0,C 180,E1 -8799.737,E2 -8799.737} C_VEL
LIN {X 0,Y 446.454,Z 294.87,A -85,B 0,C 180,E1 -8802.597,E2 -8802.597} C_VEL
LIN {X 0,Y 446.461,Z 294.871,A -85,B 0,C 180,E1 -8805.412,E2 -8805.412} C_VEL
LIN {X 0,Y 446.509,Z 294.861,A -85,B 0,C 180,E1 -8808.193,E2 -8808.193} C_VEL
LIN {X 0,Y 446.593,Z 294.852,A -85,B 0,C 180,E1 -8811.858,E2 -8811.858} C_VEL
LIN {X 0,Y 446.63,Z 294.846,A -85,B 0,C 180,E1 -8814.582,E2 -8814.582} C_VEL
LIN {X 0,Y 446.652,Z 294.843,A -85,B 0,C 180,E1 -8818.197,E2 -8818.197} C_VEL
LIN {X 0,Y 446.778,Z 294.829,A -85,B 0,C 180,E1 -8820,E2 -8820} C_VEL
LIN {X 0,Y 446.679,Z 294.84,A -85,B 0,C 180,E1 -8822.705,E2 -8822.705} C_VEL
LIN {X 0,Y 446.607,Z 294.849,A -85,B 0,C 180,E1 -8826.324,E2 -8826.324} C_VEL
LIN {X 0,Y 446.524,Z 294.86,A -85,B 0,C 180,E1 -8829.056,E2 -8829.056} C_VEL
LIN {X 0,Y 446.515,Z 294.86,A -85,B 0,C 180,E1 -8832.73,E2 -8832.73} C_VEL
LIN {X 0,Y 446.481,Z 294.866,A -85,B 0,C 180,E1 -8836.459,E2 -8836.459} C_VEL
LIN {X 0,Y 446.462,Z 294.868,A -85,B 0,C 180,E1 -8839.304,E2 -8839.304} C_VEL
LIN {X 0,Y 446.41,Z 294.879,A -85,B 0,C 180,E1 -8842.2,E2 -8842.2} C_VEL
LIN {X 0,Y 446.413,Z 294.873,A -85,B 0,C 180,E1 -8845.155,E2 -8845.155} C_VEL
LIN {X 0,Y 446.412,Z 294.881,A -85,B 0,C 180,E1 -8848.184,E2 -8848.184} C_VEL
LIN {X 0,Y 446.404,Z 294.874,A -85,B 0,C 180,E1 -8851.301,E2 -8851.301} C_VEL
LIN {X 0,Y 446.416,Z 294.878,A -85,B 0,C 180,E1 -8854.524,E2 -8854.524} C_VEL
LIN {X 0,Y 446.391,Z 294.88,A -85,B 0,C 180,E1 -8858.076,E2 -8858.076} C_VEL
LIN {X 0,Y 446.394,Z 294.875,A -85,B 0,C 180,E1 -8861.395,E2 -8861.395} C_VEL
LIN {X 0,Y 446.413,Z 294.875,A -85,B 0,C 180,E1 -8865.109,E2 -8865.109} C_VEL
LIN {X 0,Y 446.395,Z 294.883,A -85,B 0,C 180,E1 -8868.605,E2 -8868.605} C_VEL
LIN {X 0,Y 446.384,Z 294.878,A -85,B 0,C 180,E1 -8872.118,E2 -8872.118} C_VEL
LIN {X 0,Y 446.356,Z 294.881,A -85,B 0,C 180,E1 -8875.47,E2 -8875.47} C_VEL
LIN {X 0,Y 446.39,Z 294.881,A -85,B 0,C 180,E1 -8878.697,E2 -8878.697} C_VEL
LIN {X 0,Y 446.404,Z 294.874,A -85,B 0,C 180,E1 -8881.841,E2 -8881.841} C_VEL
LIN {X 0,Y 446.413,Z 294.879,A -85,B 0,C 180,E1 -8884.844,E2 -8884.844} C_VEL
LIN {X 0,Y 446.454,Z 294.868,A -85,B 0,C 180,E1 -8888.244,E2 -8888.244} C_VEL
LIN {X 0,Y 446.451,Z 294.871,A -85,B 0,C 180,E1 -8891.647,E2 -8891.647} C_VEL
LIN {X 0,Y 446.483,Z 294.864,A -85,B 0,C 180,E1 -8894.477,E2 -8894.477} C_VEL
LIN {X 0,Y 446.521,Z 294.859,A -85,B 0,C 180,E1 -8898.191,E2 -8898.191} C_VEL
LIN {X 0,Y 446.516,Z 294.862,A -85,B 0,C 180,E1 -8900.942,E2 -8900.942} C_VEL
LIN {X 0,Y 446.61,Z 294.854,A -85,B 0,C 180,E1 -8903.673,E2 -8903.673} C_VEL
LIN {X 0,Y 446.566,Z 294.855,A -85,B 0,C 180,E1 -8906.985,E2 -8906.985} C_VEL
LIN {X 0,Y 446.352,Z 294.888,A -85,B 0,C 180,E1 -8907.489,E2 -8907.489} C_VEL
LIN {X 0,Y 445.048,Z 295.049,A -85,B 0,C 180,E1 -8908.232,E2 -8908.232} C_VEL
LIN {X 0,Y 440.623,Z 295.598,A -85,B 0,C 180,E1 -8909.947,E2 -8909.947} C_VEL
LIN {X 0,Y 439.571,Z 295.726,A -85,B 0,C 180,E1 -8910.711,E2 -8910.711} C_VEL
LIN {X 0,Y 439.505,Z 295.734,A -85,B 0,C 180,E1 -8910.97,E2 -8910.97} C_VEL
LIN {X 0,Y 439.608,Z 295.72,A -85,B 0,C 180,E1 -8912.746,E2 -8912.746} C_VEL
LIN {X 0,Y 439.559,Z 295.731,A -85,B 0,C 180,E1 -8916.423,E2 -8916.423} C_VEL
LIN {X 0,Y 439.493,Z 295.74,A -85,B 0,C 180,E1 -8919.198,E2 -8919.198} C_VEL
LIN {X 0,Y 439.487,Z 295.764,A -85,B 0,C 180,E1 -8920.36,E2 -8920.36} C_VEL
LIN {X 0,Y 440.85,Z 303.691,A -85,B 0,C 180,E1 -8922.191,E2 -8922.191} C_VEL
LIN {X 0,Y 440.68,Z 311.926,A -85,B 0,C 180,E1 -8923.982,E2 -8923.982} C_VEL
LIN {X 0,Y 444.177,Z 329.405,A -85,B 0,C 180,E1 -8924.435,E2 -8924.435} C_VEL
LIN {X 0,Y 443.128,Z 418.919,A -85,B 0,C 180,E1 -8925.933,E2 -8925.933} C_VEL
LIN {X 0,Y 442.846,Z 432.699,A -85,B 0,C 180,E1 -8926.357,E2 -8926.357} C_VEL
LIN {X 0,Y 442.44,Z 444.463,A -85,B 0,C 180,E1 -8926.89,E2 -8926.89} C_VEL
LIN {X 0,Y 441.934,Z 455.927,A -85,B 0,C 180,E1 -8927.583,E2 -8927.583} C_VEL
LIN {X 0,Y 441.387,Z 466.966,A -85,B 0,C 180,E1 -8928.445,E2 -8928.445} C_VEL
LIN {X 0,Y 440.715,Z 477.222,A -85,B 0,C 180,E1 -8929.44,E2 -8929.44} C_VEL
LIN {X 0,Y 440.201,Z 486.567,A -85,B 0,C 180,E1 -8930.558,E2 -8930.558} C_VEL
LIN {X 0,Y 439.719,Z 494.926,A -85,B 0,C 180,E1 -8931.782,E2 -8931.782} C_VEL
LIN {X 0,Y 439.269,Z 502.111,A -85,B 0,C 180,E1 -8933.073,E2 -8933.073} C_VEL
LIN {X 0,Y 438.882,Z 508.881,A -85,B 0,C 180,E1 -8934.599,E2 -8934.599} C_VEL
LIN {X 0,Y 438.641,Z 514.373,A -85,B 0,C 180,E1 -8936.201,E2 -8936.201} C_VEL
LIN {X 0,Y 438.417,Z 518.159,A -85,B 0,C 180,E1 -8937.697,E2 -8937.697} C_VEL
LIN {X 0,Y 438.279,Z 520.087,A -85,B 0,C 180,E1 -8938.749,E2 -8938.749} C_VEL
LIN {X 0,Y 438.221,Z 521.707,A -85,B 0,C 180,E1 -8939.999,E2 -8939.999} C_VEL
LIN {X 0,Y 438.189,Z 522.704,A -85,B 0,C 180,E1 -8941.782,E2 -8941.782} C_VEL
LIN {X 0,Y 438.195,Z 522.294,A -85,B 0,C 180,E1 -8943.487,E2 -8943.487} C_VEL
LIN {X 0,Y 438.289,Z 520.382,A -85,B 0,C 180,E1 -8945.252,E2 -8945.252} C_VEL
LIN {X 0,Y 438.493,Z 517.599,A -85,B 0,C 180,E1 -8946.738,E2 -8946.738} C_VEL
LIN {X 0,Y 438.69,Z 513.487,A -85,B 0,C 180,E1 -8948.279,E2 -8948.279} C_VEL
LIN {X 0,Y 438.978,Z 508.025,A -85,B 0,C 180,E1 -8949.814,E2 -8949.814} C_VEL
LIN {X 0,Y 439.369,Z 501.439,A -85,B 0,C 180,E1 -8951.254,E2 -8951.254} C_VEL
LIN {X 0,Y 439.869,Z 493.12,A -85,B 0,C 180,E1 -8952.696,E2 -8952.696} C_VEL
LIN {X 0,Y 440.455,Z 484.428,A -85,B 0,C 180,E1 -8953.913,E2 -8953.913} C_VEL
LIN {X 0,Y 441.09,Z 475.022,A -85,B 0,C 180,E1 -8954.986,E2 -8954.986} C_VEL
LIN {X 0,Y 441.587,Z 465.261,A -85,B 0,C 180,E1 -8955.896,E2 -8955.896} C_VEL
LIN {X 0,Y 442.277,Z 452.915,A -85,B 0,C 180,E1 -8956.803,E2 -8956.803} C_VEL
LIN {X 0,Y 442.784,Z 440.99,A -85,B 0,C 180,E1 -8957.474,E2 -8957.474} C_VEL
LIN {X 0,Y 443.166,Z 428.139,A -85,B 0,C 180,E1 -8957.989,E2 -8957.989} C_VEL
LIN {X 0,Y 443.448,Z 414.437,A -85,B 0,C 180,E1 -8958.335,E2 -8958.335} C_VEL
LIN {X 0,Y 444.362,Z 329.054,A -85,B 0,C 180,E1 -8959.761,E2 -8959.761} C_VEL
LIN {X 0,Y 440.774,Z 311.601,A -85,B 0,C 180,E1 -8960.247,E2 -8960.247} C_VEL
LIN {X 0,Y 440.881,Z 303.297,A -85,B 0,C 180,E1 -8961.851,E2 -8961.851} C_VEL
LIN {X 0,Y 439.344,Z 295.758,A -85,B 0,C 180,E1 -8963.446,E2 -8963.446} C_VEL
LIN {X 0,Y 439.357,Z 295.76,A -85,B 0,C 180,E1 -8966.272,E2 -8966.272} C_VEL
LIN {X 0,Y 439.371,Z 295.756,A -85,B 0,C 180,E1 -8969.729,E2 -8969.729} C_VEL
LIN {X 0,Y 439.401,Z 295.757,A -85,B 0,C 180,E1 -8972.365,E2 -8972.365} C_VEL
LIN {X 0,Y 439.369,Z 295.758,A -85,B 0,C 180,E1 -8975.733,E2 -8975.733} C_VEL
LIN {X 0,Y 439.339,Z 295.759,A -85,B 0,C 180,E1 -8979.395,E2 -8979.395} C_VEL
LIN {X 0,Y 439.381,Z 295.756,A -85,B 0,C 180,E1 -8982.307,E2 -8982.307} C_VEL
LIN {X 0,Y 439.395,Z 295.751,A -85,B 0,C 180,E1 -8985.172,E2 -8985.172} C_VEL
LIN {X 0,Y 439.433,Z 295.745,A -85,B 0,C 180,E1 -8988,E2 -8988} C_VEL
LIN {X 0,Y 439.496,Z 295.735,A -85,B 0,C 180,E1 -8991.725,E2 -8991.725} C_VEL
LIN {X 0,Y 439.565,Z 295.731,A -85,B 0,C 180,E1 -8994.495,E2 -8994.495} C_VEL
LIN {X 0,Y 439.584,Z 295.725,A -85,B 0,C 180,E1 -8998.168,E2 -8998.168} C_VEL
LIN {X 0,Y 439.709,Z 295.704,A -85,B 0,C 180,E1 -9000,E2 -9000} C_VEL
LIN {X 0,Y 439.611,Z 295.726,A -85,B 0,C 180,E1 -9002.749,E2 -9002.749} C_VEL
LIN {X 0,Y 439.568,Z 295.728,A -85,B 0,C 180,E1 -9006.426,E2 -9006.426} C_VEL
LIN {X 0,Y 439.455,Z 295.747,A -85,B 0,C 180,E1 -9009.203,E2 -9009.203} C_VEL
LIN {X 0,Y 439.454,Z 295.738,A -85,B 0,C 180,E1 -9012.728,E2 -9012.728} C_VEL
LIN {X 0,Y 439.411,Z 295.741,A -85,B 0,C 180,E1 -9016.356,E2 -9016.356} C_VEL
LIN {X 0,Y 439.387,Z 295.746,A -85,B 0,C 180,E1 -9019.627,E2 -9019.627} C_VEL
LIN {X 0,Y 439.34,Z 295.754,A -85,B 0,C 180,E1 -9022.577,E2 -9022.577} C_VEL
LIN {X 0,Y 439.371,Z 295.755,A -85,B 0,C 180,E1 -9025.587,E2 -9025.587} C_VEL
LIN {X 0,Y 439.382,Z 295.745,A -85,B 0,C 180,E1 -9028.676,E2 -9028.676} C_VEL
LIN {X 0,Y 439.334,Z 295.757,A -85,B 0,C 180,E1 -9031.864,E2 -9031.864} C_VEL
LIN {X 0,Y 439.364,Z 295.755,A -85,B 0,C 180,E1 -9035.159,E2 -9035.159} C_VEL
LIN {X 0,Y 439.405,Z 295.746,A -85,B 0,C 180,E1 -9038.593,E2 -9038.593} C_VEL
LIN {X 0,Y 439.372,Z 295.755,A -85,B 0,C 180,E1 -9041.263,E2 -9041.263} C_VEL
LIN {X 0,Y 439.379,Z 295.754,A -85,B 0,C 180,E1 -9044.732,E2 -9044.732} C_VEL
LIN {X 0,Y 439.385,Z 295.758,A -85,B 0,C 180,E1 -9047.802,E2 -9047.802} C_VEL
LIN {X 0,Y 439.428,Z 295.749,A -85,B 0,C 180,E1 -9050.235,E2 -9050.235} C_VEL
LIN {X 0,Y 439.355,Z 295.757,A -85,B 0,C 180,E1 -9053.718,E2 -9053.718} C_VEL
LIN {X 0,Y 439.353,Z 295.759,A -85,B 0,C 180,E1 -9057.058,E2 -9057.058} C_VEL
LIN {X 0,Y 439.38,Z 295.758,A -85,B 0,C 180,E1 -9060.28,E2 -9060.28} C_VEL
LIN {X 0,Y 439.467,Z 295.804,A -85,B 0,C 180,E1 -9063.212,E2 -9063.212} C_VEL
LIN {X 0,Y 441.844,Z 307.689,A -85,B 0,C 180,E1 -9065.577,E2 -9065.577} C_VEL
LIN {X 0,Y 441.95,Z 311.72,A -85,B 0,C 180,E1 -9066.331,E2 -9066.331} C_VEL
LIN {X 0,Y 441.106,Z 327.754,A -85,B 0,C 180,E1 -9069.242,E2 -9069.242} C_VEL
LIN {X 0,Y 440.445,Z 342.012,A -85,B 0,C 180,E1 -9071.802,E2 -9071.802} C_VEL
LIN {X 0,Y 444.093,Z 366.586,A -85,B 0,C 180,E1 -9072.387,E2 -9072.387} C_VEL
LIN {X 0,Y 443.161,Z 450.716,A -85,B 0,C 180,E1 -9073.803,E2 -9073.803} C_VEL
LIN {X 0,Y 442.746,Z 463.915,A -85,B 0,C 180,E1 -9074.201,E2 -9074.201} C_VEL
LIN {X 0,Y 442.181,Z 476.07,A -85,B 0,C 180,E1 -9074.742,E2 -9074.742} C_VEL
LIN {X 0,Y 441.548,Z 488.371,A -85,B 0,C 180,E1 -9075.486,E2 -9075.486} C_VEL
LIN {X 0,Y 440.984,Z 499.401,A -85,B 0,C 180,E1 -9076.354,E2 -9076.354} C_VEL
LIN {X 0,Y 440.295,Z 510.49,A -85,B 0,C 180,E1 -9077.443,E2 -9077.443} C_VEL
LIN {X 0,Y 439.795,Z 519.071,A -85,B 0,C 180,E1 -9078.481,E2 -9078.481} C_VEL
LIN {X 0,Y 439.267,Z 526.992,A -85,B 0,C 180,E1 -9079.634,E2 -9079.634} C_VEL
LIN {X 0,Y 438.869,Z 534.735,A -85,B 0,C 180,E1 -9081.021,E2 -9081.021} C_VEL
LIN {X 0,Y 438.548,Z 541.881,A -85,B 0,C 180,E1 -9082.638,E2 -9082.638} C_VEL
LIN {X 0,Y 438.379,Z 546.519,A -85,B 0,C 180,E1 -9083.984,E2 -9083.984} C_VEL
LIN {X 0,Y 438.34,Z 550.279,A -85,B 0,C 180,E1 -9085.405,E2 -9085.405} C_VEL
LIN {X 0,Y 438.282,Z 552.153,A -85,B 0,C 180,E1 -9086.326,E2 -9086.326} C_VEL
LIN {X 0,Y 438.34,Z 553.562,A -85,B 0,C 180,E1 -9087.246,E2 -9087.246} C_VEL
LIN {X 0,Y 438.277,Z 555.182,A -85,B 0,C 180,E1 -9089.084,E2 -9089.084} C_VEL
LIN {X 0,Y 438.281,Z 555.394,A -85,B 0,C 180,E1 -9090.003,E2 -9090.003} C_VEL
LIN {X 0,Y 438.296,Z 554.556,A -85,B 0,C 180,E1 -9091.841,E2 -9091.841} C_VEL
LIN {X 0,Y 438.341,Z 553.551,A -85,B 0,C 180,E1 -9092.76,E2 -9092.76} C_VEL
LIN {X 0,Y 438.284,Z 552.125,A -85,B 0,C 180,E1 -9093.68,E2 -9093.68} C_VEL
LIN {X 0,Y 438.384,Z 549.155,A -85,B 0,C 180,E1 -9095.061,E2 -9095.061} C_VEL
LIN {X 0,Y 438.45,Z 545.126,A -85,B 0,C 180,E1 -9096.445,E2 -9096.445} C_VEL
LIN {X 0,Y 438.678,Z 538.922,A -85,B 0,C 180,E1 -9098.061,E2 -9098.061} C_VEL
LIN {X 0,Y 438.97,Z 532.154,A -85,B 0,C 180,E1 -9099.448,E2 -9099.448} C_VEL
LIN {X 0,Y 439.423,Z 523.755,A -85,B 0,C 180,E1 -9100.834,E2 -9100.834} C_VEL
LIN {X 0,Y 439.988,Z 515.099,A -85,B 0,C 180,E1 -9101.987,E2 -9101.987} C_VEL
LIN {X 0,Y 440.54,Z 505.32,A -85,B 0,C 180,E1 -9103.053,E2 -9103.053} C_VEL
LIN {X 0,Y 441.172,Z 493.84,A -85,B 0,C 180,E1 -9104.062,E2 -9104.062} C_VEL
LIN {X 0,Y 441.822,Z 482.095,A -85,B 0,C 180,E1 -9104.864,E2 -9104.864} C_VEL
LIN {X 0,Y 442.372,Z 469.895,A -85,B 0,C 180,E1 -9105.494,E2 -9105.494} C_VEL
LIN {X 0,Y 442.85,Z 456.606,A -85,B 0,C 180,E1 -9105.979,E2 -9105.979} C_VEL
LIN {X 0,Y 443.232,Z 441.786,A -85,B 0,C 180,E1 -9106.289,E2 -9106.289} C_VEL
LIN {X 0,Y 443.881,Z 365.652,A -85,B 0,C 180,E1 -9107.553,E2 -9107.553} C_VEL
LIN {X 0,Y 440.412,Z 342.768,A -85,B 0,C 180,E1 -9108.084,E2 -9108.084} C_VEL
LIN {X 0,Y 441.257,Z 326.915,A -85,B 0,C 180,E1 -9111.001,E2 -9111.001} C_VEL
LIN {X 0,Y 442.172,Z 311.285,A -85,B 0,C 180,E1 -9113.912,E2 -9113.912} C_VEL
LIN {X 0,Y 441.38,Z 305.262,A -85,B 0,C 180,E1 -9115.106,E2 -9115.106} C_VEL
LIN {X 0,Y 439.479,Z 295.744,A -85,B 0,C 180,E1 -9117.083,E2 -9117.083} C_VEL
LIN {X 0,Y 439.385,Z 295.757,A -85,B 0,C 180,E1 -9120.261,E2 -9120.261} C_VEL
LIN {X 0,Y 439.401,Z 295.749,A -85,B 0,C 180,E1 -9123.724,E2 -9123.724} C_VEL
LIN {X 0,Y 439.351,Z 295.753,A -85,B 0,C 180,E1 -9126.887,E2 -9126.887} C_VEL
LIN {X 0,Y 439.405,Z 295.748,A -85,B 0,C 180,E1 -9129.849,E2 -9129.849} C_VEL
LIN {X 0,Y 439.383,Z 295.753,A -85,B 0,C 180,E1 -9132.627,E2 -9132.627} C_VEL
LIN {X 0,Y 439.4,Z 295.747,A -85,B 0,C 180,E1 -9135.27,E2 -9135.27} C_VEL
LIN {X 0,Y 439.389,Z 295.753,A -85,B 0,C 180,E1 -9138.743,E2 -9138.743} C_VEL
LIN {X 0,Y 439.376,Z 295.749,A -85,B 0,C 180,E1 -9141.607,E2 -9141.607} C_VEL
LIN {X 0,Y 439.398,Z 295.752,A -85,B 0,C 180,E1 -9144.844,E2 -9144.844} C_VEL
LIN {X 0,Y 439.37,Z 295.752,A -85,B 0,C 180,E1 -9148.139,E2 -9148.139} C_VEL
LIN {X 0,Y 439.429,Z 295.743,A -85,B 0,C 180,E1 -9151.598,E2 -9151.598} C_VEL
LIN {X 0,Y 439.401,Z 295.749,A -85,B 0,C 180,E1 -9154.415,E2 -9154.415} C_VEL
LIN {X 0,Y 439.359,Z 295.754,A -85,B 0,C 180,E1 -9157.424,E2 -9157.424} C_VEL
LIN {X 0,Y 439.436,Z 295.745,A -85,B 0,C 180,E1 -9160.663,E2 -9160.663} C_VEL
LIN {X 0,Y 439.455,Z 295.74,A -85,B 0,C 180,E1 -9164.224,E2 -9164.224} C_VEL
LIN {X 0,Y 439.476,Z 295.737,A -85,B 0,C 180,E1 -9168.001,E2 -9168.001} C_VEL
LIN {X 0,Y 439.541,Z 295.732,A -85,B 0,C 180,E1 -9171.726,E2 -9171.726} C_VEL
LIN {X 0,Y 439.606,Z 295.721,A -85,B 0,C 180,E1 -9174.496,E2 -9174.496} C_VEL
LIN {X 0,Y 439.623,Z 295.719,A -85,B 0,C 180,E1 -9178.168,E2 -9178.168} C_VEL
LIN {X 0,Y 439.748,Z 295.705,A -85,B 0,C 180,E1 -9180,E2 -9180} C_VEL
LIN {X 0,Y 439.629,Z 295.718,A -85,B 0,C 180,E1 -9182.749,E2 -9182.749} C_VEL
LIN {X 0,Y 439.559,Z 295.727,A -85,B 0,C 180,E1 -9186.426,E2 -9186.426} C_VEL
LIN {X 0,Y 439.487,Z 295.738,A -85,B 0,C 180,E1 -9189.202,E2 -9189.202} C_VEL
LIN {X 0,Y 439.458,Z 295.739,A -85,B 0,C 180,E1 -9192.938,E2 -9192.938} C_VEL
LIN {X 0,Y 439.439,Z 295.744,A -85,B 0,C 180,E1 -9196.348,E2 -9196.348} C_VEL
LIN {X 0,Y 439.396,Z 295.751,A -85,B 0,C 180,E1 -9199.627,E2 -9199.627} C_VEL
LIN {X 0,Y 439.355,Z 295.754,A -85,B 0,C 180,E1 -9202.576,E2 -9202.576} C_VEL
LIN {X 0,Y 439.36,Z 295.754,A -85,B 0,C 180,E1 -9205.588,E2 -9205.588} C_VEL
LIN {X 0,Y 439.377,Z 295.751,A -85,B 0,C 180,E1 -9208.676,E2 -9208.676} C_VEL
LIN {X 0,Y 439.359,Z 295.757,A -85,B 0,C 180,E1 -9212.029,E2 -9212.029} C_VEL
LIN {X 0,Y 439.383,Z 295.749,A -85,B 0,C 180,E1 -9215.339,E2 -9215.339} C_VEL
LIN {X 0,Y 439.346,Z 295.759,A -85,B 0,C 180,E1 -9218.599,E2 -9218.599} C_VEL
LIN {X 0,Y 439.343,Z 295.758,A -85,B 0,C 180,E1 -9222.211,E2 -9222.211} C_VEL
LIN {X 0,Y 439.367,Z 295.751,A -85,B 0,C 180,E1 -9225.266,E2 -9225.266} C_VEL
LIN {X 0,Y 439.358,Z 295.759,A -85,B 0,C 180,E1 -9228.748,E2 -9228.748} C_VEL
LIN {X 0,Y 439.35,Z 295.753,A -85,B 0,C 180,E1 -9231.612,E2 -9231.612} C_VEL
LIN {X 0,Y 439.334,Z 295.763,A -85,B 0,C 180,E1 -9234.837,E2 -9234.837} C_VEL
LIN {X 0,Y 439.342,Z 295.754,A -85,B 0,C 180,E1 -9238.136,E2 -9238.136} C_VEL
LIN {X 0,Y 439.381,Z 295.752,A -85,B 0,C 180,E1 -9241.323,E2 -9241.323} C_VEL
LIN {X 0,Y 439.348,Z 295.754,A -85,B 0,C 180,E1 -9244.41,E2 -9244.41} C_VEL
LIN {X 0,Y 439.367,Z 295.754,A -85,B 0,C 180,E1 -9247.423,E2 -9247.423} C_VEL
LIN {X 0,Y 439.447,Z 295.743,A -85,B 0,C 180,E1 -9250.662,E2 -9250.662} C_VEL
LIN {X 0,Y 439.451,Z 295.74,A -85,B 0,C 180,E1 -9254.222,E2 -9254.222} C_VEL
LIN {X 0,Y 439.488,Z 295.736,A -85,B 0,C 180,E1 -9257.999,E2 -9257.999} C_VEL
LIN {X 0,Y 439.485,Z 295.74,A -85,B 0,C 180,E1 -9261.723,E2 -9261.723} C_VEL
LIN {X 0,Y 439.601,Z 295.721,A -85,B 0,C 180,E1 -9264.493,E2 -9264.493} C_VEL
LIN {X 0,Y 439.629,Z 295.719,A -85,B 0,C 180,E1 -9268.165,E2 -9268.165} C_VEL
LIN {X 0,Y 439.69,Z 295.714,A -85,B 0,C 180,E1 -9269.997,E2 -9269.997} C_VEL
LIN {X 0,Y 439.505,Z 295.734,A -85,B 0,C 180,E1 -9270.97,E2 -9270.97} C_VEL
LIN {X 0,Y 438.861,Z 295.821,A -85,B 0,C 180,E1 -9271.735,E2 -9271.735} C_VEL
LIN {X 0,Y 435.924,Z 296.18,A -85,B 0,C 180,E1 -9272.975,E2 -9272.975} C_VEL
LIN {X 0,Y 433.464,Z 296.492,A -85,B 0,C 180,E1 -9273.977,E2 -9273.977} C_VEL
LIN {X 0,Y 432.479,Z 296.61,A -85,B 0,C 180,E1 -9274.752,E2 -9274.752} C_VEL
LIN {X 0,Y 432.44,Z 296.614,A -85,B 0,C 180,E1 -9275.014,E2 -9275.014} C_VEL
LIN {X 0,Y 432.504,Z 296.613,A -85,B 0,C 180,E1 -9277.595,E2 -9277.595} C_VEL
LIN {X 0,Y 432.446,Z 296.713,A -85,B 0,C 180,E1 -9280.176,E2 -9280.176} C_VEL
LIN {X 0,Y 433.913,Z 305.153,A -85,B 0,C 180,E1 -9282.151,E2 -9282.151} C_VEL
LIN {X 0,Y 433.737,Z 312.164,A -85,B 0,C 180,E1 -9283.695,E2 -9283.695} C_VEL
LIN {X 0,Y 437.384,Z 330.296,A -85,B 0,C 180,E1 -9284.176,E2 -9284.176} C_VEL
LIN {X 0,Y 436.284,Z 420.136,A -85,B 0,C 180,E1 -9285.713,E2 -9285.713} C_VEL
LIN {X 0,Y 435.97,Z 433.543,A -85,B 0,C 180,E1 -9286.141,E2 -9286.141} C_VEL
LIN {X 0,Y 435.556,Z 445.462,A -85,B 0,C 180,E1 -9286.699,E2 -9286.699} C_VEL
LIN {X 0,Y 434.994,Z 457.264,A -85,B 0,C 180,E1 -9287.442,E2 -9287.442} C_VEL
LIN {X 0,Y 434.333,Z 468.894,A -85,B 0,C 180,E1 -9288.388,E2 -9288.388} C_VEL
LIN {X 0,Y 433.701,Z 478.832,A -85,B 0,C 180,E1 -9289.398,E2 -9289.398} C_VEL
LIN {X 0,Y 433.063,Z 488.852,A -85,B 0,C 180,E1 -9290.664,E2 -9290.664} C_VEL
LIN {X 0,Y 432.598,Z 496.981,A -85,B 0,C 180,E1 -9291.937,E2 -9291.937} C_VEL
LIN {X 0,Y 432.107,Z 504.928,A -85,B 0,C 180,E1 -9293.478,E2 -9293.478} C_VEL
LIN {X 0,Y 431.729,Z 511.15,A -85,B 0,C 180,E1 -9295.035,E2 -9295.035} C_VEL
LIN {X 0,Y 431.535,Z 515.403,A -85,B 0,C 180,E1 -9296.397,E2 -9296.397} C_VEL
LIN {X 0,Y 431.264,Z 519.498,A -85,B 0,C 180,E1 -9298.197,E2 -9298.197} C_VEL
LIN {X 0,Y 431.163,Z 521.164,A -85,B 0,C 180,E1 -9299.269,E2 -9299.269} C_VEL
LIN {X 0,Y 431.103,Z 522.294,A -85,B 0,C 180,E1 -9300.35,E2 -9300.35} C_VEL
LIN {X 0,Y 431.081,Z 523.013,A -85,B 0,C 180,E1 -9302.03,E2 -9302.03} C_VEL
LIN {X 0,Y 431.1,Z 522.386,A -85,B 0,C 180,E1 -9303.754,E2 -9303.754} C_VEL
LIN {X 0,Y 431.216,Z 520.485,A -85,B 0,C 180,E1 -9305.422,E2 -9305.422} C_VEL
LIN {X 0,Y 431.456,Z 517.344,A -85,B 0,C 180,E1 -9307.056,E2 -9307.056} C_VEL
LIN {X 0,Y 431.671,Z 513.114,A -85,B 0,C 180,E1 -9308.603,E2 -9308.603} C_VEL
LIN {X 0,Y 431.978,Z 507.593,A -85,B 0,C 180,E1 -9310.123,E2 -9310.123} C_VEL
LIN {X 0,Y 432.443,Z 500.633,A -85,B 0,C 180,E1 -9311.618,E2 -9311.618} C_VEL
LIN {X 0,Y 432.981,Z 492.125,A -85,B 0,C 180,E1 -9313.078,E2 -9313.078} C_VEL
LIN {X 0,Y 433.656,Z 482.759,A -85,B 0,C 180,E1 -9314.355,E2 -9314.355} C_VEL
LIN {X 0,Y 434.381,Z 472.06,A -85,B 0,C 180,E1 -9315.527,E2 -9315.527} C_VEL
LIN {X 0,Y 434.955,Z 461.894,A -85,B 0,C 180,E1 -9316.425,E2 -9316.425} C_VEL
LIN {X 0,Y 435.538,Z 449.922,A -85,B 0,C 180,E1 -9317.255,E2 -9317.255} C_VEL
LIN {X 0,Y 436.144,Z 437.159,A -85,B 0,C 180,E1 -9317.914,E2 -9317.914} C_VEL
LIN {X 0,Y 436.497,Z 424.297,A -85,B 0,C 180,E1 -9318.381,E2 -9318.381} C_VEL
LIN {X 0,Y 436.76,Z 407.934,A -85,B 0,C 180,E1 -9318.72,E2 -9318.72} C_VEL
LIN {X 0,Y 437.7,Z 330.238,A -85,B 0,C 180,E1 -9320.039,E2 -9320.039} C_VEL
LIN {X 0,Y 433.876,Z 311.872,A -85,B 0,C 180,E1 -9320.56,E2 -9320.56} C_VEL
LIN {X 0,Y 433.918,Z 304.462,A -85,B 0,C 180,E1 -9322.014,E2 -9322.014} C_VEL
LIN {X 0,Y 432.325,Z 296.633,A -85,B 0,C 180,E1 -9323.677,E2 -9323.677} C_VEL
LIN {X 0,Y 432.3,Z 296.639,A -85,B 0,C 180,E1 -9326.444,E2 -9326.444} C_VEL
LIN {X 0,Y 432.353,Z 296.63,A -85,B 0,C 180,E1 -9329.741,E2 -9329.741} C_VEL
LIN {X 0,Y 432.356,Z 296.63,A -85,B 0,C 180,E1 -9333.369,E2 -9333.369} C_VEL
LIN {X 0,Y 432.325,Z 296.638,A -85,B 0,C 180,E1 -9336.021,E2 -9336.021} C_VEL
LIN {X 0,Y 432.301,Z 296.637,A -85,B 0,C 180,E1 -9339.043,E2 -9339.043} C_VEL
LIN {X 0,Y 432.328,Z 296.631,A -85,B 0,C 180,E1 -9342.009,E2 -9342.009} C_VEL
LIN {X 0,Y 432.344,Z 296.631,A -85,B 0,C 180,E1 -9344.925,E2 -9344.925} C_VEL
LIN {X 0,Y 432.408,Z 296.619,A -85,B 0,C 180,E1 -9347.802,E2 -9347.802} C_VEL
LIN {X 0,Y 432.44,Z 296.614,A -85,B 0,C 180,E1 -9351.589,E2 -9351.589} C_VEL
LIN {X 0,Y 432.542,Z 296.605,A -85,B 0,C 180,E1 -9354.405,E2 -9354.405} C_VEL
LIN {X 0,Y 432.554,Z 296.601,A -85,B 0,C 180,E1 -9358.138,E2 -9358.138} C_VEL
LIN {X 0,Y 432.679,Z 296.579,A -85,B 0,C 180,E1 -9360,E2 -9360} C_VEL
LIN {X 0,Y 432.561,Z 296.603,A -85,B 0,C 180,E1 -9362.794,E2 -9362.794} C_VEL
LIN {X 0,Y 432.523,Z 296.607,A -85,B 0,C 180,E1 -9366.531,E2 -9366.531} C_VEL
LIN {X 0,Y 432.398,Z 296.624,A -85,B 0,C 180,E1 -9369.354,E2 -9369.354} C_VEL
LIN {X 0,Y 432.395,Z 296.618,A -85,B 0,C 180,E1 -9372.813,E2 -9372.813} C_VEL
LIN {X 0,Y 432.374,Z 296.618,A -85,B 0,C 180,E1 -9376.485,E2 -9376.485} C_VEL
LIN {X 0,Y 432.335,Z 296.622,A -85,B 0,C 180,E1 -9379.961,E2 -9379.961} C_VEL
LIN {X 0,Y 432.289,Z 296.635,A -85,B 0,C 180,E1 -9382.966,E2 -9382.966} C_VEL
LIN {X 0,Y 432.325,Z 296.628,A -85,B 0,C 180,E1 -9386.035,E2 -9386.035} C_VEL
LIN {X 0,Y 432.31,Z 296.631,A -85,B 0,C 180,E1 -9389.19,E2 -9389.19} C_VEL
LIN {X 0,Y 432.285,Z 296.632,A -85,B 0,C 180,E1 -9392.297,E2 -9392.297} C_VEL
LIN {X 0,Y 432.303,Z 296.631,A -85,B 0,C 180,E1 -9394.681,E2 -9394.681} C_VEL
LIN {X 0,Y 432.348,Z 296.627,A -85,B 0,C 180,E1 -9398.149,E2 -9398.149} C_VEL
LIN {X 0,Y 432.34,Z 296.633,A -85,B 0,C 180,E1 -9401.612,E2 -9401.612} C_VEL
LIN {X 0,Y 432.348,Z 296.631,A -85,B 0,C 180,E1 -9404.346,E2 -9404.346} C_VEL
LIN {X 0,Y 432.337,Z 296.632,A -85,B 0,C 180,E1 -9407.013,E2 -9407.013} C_VEL
LIN {X 0,Y 432.334,Z 296.635,A -85,B 0,C 180,E1 -9409.821,E2 -9409.821} C_VEL
LIN {X 0,Y 432.295,Z 296.634,A -85,B 0,C 180,E1 -9413.028,E2 -9413.028} C_VEL
LIN {X 0,Y 432.339,Z 296.633,A -85,B 0,C 180,E1 -9416.001,E2 -9416.001} C_VEL
LIN {X 0,Y 432.378,Z 296.634,A -85,B 0,C 180,E1 -9419.749,E2 -9419.749} C_VEL
LIN {X 0,Y 432.456,Z 296.757,A -85,B 0,C 180,E1 -9422.969,E2 -9422.969} C_VEL
LIN {X 0,Y 435.065,Z 310.131,A -85,B 0,C 180,E1 -9425.679,E2 -9425.679} C_VEL
LIN {X 0,Y 434.442,Z 323.516,A -85,B 0,C 180,E1 -9428.161,E2 -9428.161} C_VEL
LIN {X 0,Y 433.523,Z 341.696,A -85,B 0,C 180,E1 -9431.483,E2 -9431.483} C_VEL
LIN {X 0,Y 437.339,Z 367.073,A -85,B 0,C 180,E1 -9432.105,E2 -9432.105} C_VEL
LIN {X 0,Y 436.355,Z 450.723,A -85,B 0,C 180,E1 -9433.543,E2 -9433.543} C_VEL
LIN {X 0,Y 435.859,Z 464.583,A -85,B 0,C 180,E1 -9433.975,E2 -9433.975} C_VEL
LIN {X 0,Y 435.282,Z 477.048,A -85,B 0,C 180,E1 -9434.554,E2 -9434.554} C_VEL
LIN {X 0,Y 434.665,Z 488.19,A -85,B 0,C 180,E1 -9435.251,E2 -9435.251} C_VEL
LIN {X 0,Y 434.03,Z 499.689,A -85,B 0,C 180,E1 -9436.175,E2 -9436.175} C_VEL
LIN {X 0,Y 433.314,Z 510.281,A -85,B 0,C 180,E1 -9437.237,E2 -9437.237} C_VEL
LIN {X 0,Y 432.812,Z 518.854,A -85,B 0,C 180,E1 -9438.293,E2 -9438.293} C_VEL
LIN {X 0,Y 432.237,Z 526.766,A -85,B 0,C 180,E1 -9439.464,E2 -9439.464} C_VEL
LIN {X 0,Y 431.817,Z 534.5,A -85,B 0,C 180,E1 -9440.873,E2 -9440.873} C_VEL
LIN {X 0,Y 431.494,Z 541.643,A -85,B 0,C 180,E1 -9442.517,E2 -9442.517} C_VEL
LIN {X 0,Y 431.278,Z 546.712,A -85,B 0,C 180,E1 -9444.027,E2 -9444.027} C_VEL
LIN {X 0,Y 431.269,Z 550.029,A -85,B 0,C 180,E1 -9445.33,E2 -9445.33} C_VEL
LIN {X 0,Y 431.188,Z 551.898,A -85,B 0,C 180,E1 -9446.265,E2 -9446.265} C_VEL
LIN {X 0,Y 431.236,Z 553.305,A -85,B 0,C 180,E1 -9447.201,E2 -9447.201} C_VEL
LIN {X 0,Y 431.218,Z 554.309,A -85,B 0,C 180,E1 -9448.135,E2 -9448.135} C_VEL
LIN {X 0,Y 431.192,Z 554.921,A -85,B 0,C 180,E1 -9449.069,E2 -9449.069} C_VEL
LIN {X 0,Y 431.194,Z 555.129,A -85,B 0,C 180,E1 -9450.003,E2 -9450.003} C_VEL
LIN {X 0,Y 431.219,Z 554.286,A -85,B 0,C 180,E1 -9451.871,E2 -9451.871} C_VEL
LIN {X 0,Y 431.238,Z 553.276,A -85,B 0,C 180,E1 -9452.805,E2 -9452.805} C_VEL
LIN {X 0,Y 431.19,Z 551.845,A -85,B 0,C 180,E1 -9453.741,E2 -9453.741} C_VEL
LIN {X 0,Y 431.295,Z 548.868,A -85,B 0,C 180,E1 -9455.145,E2 -9455.145} C_VEL
LIN {X 0,Y 431.378,Z 544.829,A -85,B 0,C 180,E1 -9456.551,E2 -9456.551} C_VEL
LIN {X 0,Y 431.609,Z 538.608,A -85,B 0,C 180,E1 -9458.194,E2 -9458.194} C_VEL
LIN {X 0,Y 431.92,Z 531.824,A -85,B 0,C 180,E1 -9459.603,E2 -9459.603} C_VEL
LIN {X 0,Y 432.417,Z 523.4,A -85,B 0,C 180,E1 -9461.012,E2 -9461.012} C_VEL
LIN {X 0,Y 433.003,Z 514.718,A -85,B 0,C 180,E1 -9462.183,E2 -9462.183} C_VEL
LIN {X 0,Y 433.633,Z 504.363,A -85,B 0,C 180,E1 -9463.321,E2 -9463.321} C_VEL
LIN {X 0,Y 434.256,Z 493.402,A -85,B 0,C 180,E1 -9464.291,E2 -9464.291} C_VEL
LIN {X 0,Y 434.951,Z 481.589,A -85,B 0,C 180,E1 -9465.105,E2 -9465.105} C_VEL
LIN {X 0,Y 435.495,Z 469.312,A -85,B 0,C 180,E1 -9465.745,E2 -9465.745} C_VEL
LIN {X 0,Y 436.035,Z 455.873,A -85,B 0,C 180,E1 -9466.235,E2 -9466.235} C_VEL
LIN {X 0,Y 436.382,Z 440.669,A -85,B 0,C 180,E1 -9466.552,E2 -9466.552} C_VEL
LIN {X 0,Y 436.986,Z 365.578,A -85,B 0,C 180,E1 -9467.823,E2 -9467.823} C_VEL
LIN {X 0,Y 433.48,Z 342.461,A -85,B 0,C 180,E1 -9468.383,E2 -9468.383} C_VEL
LIN {X 0,Y 434.372,Z 326.598,A -85,B 0,C 180,E1 -9471.35,E2 -9471.35} C_VEL
LIN {X 0,Y 435.233,Z 312.28,A -85,B 0,C 180,E1 -9474.064,E2 -9474.064} C_VEL
LIN {X 0,Y 434.015,Z 304.293,A -85,B 0,C 180,E1 -9475.687,E2 -9475.687} C_VEL
LIN {X 0,Y 432.447,Z 296.619,A -85,B 0,C 180,E1 -9477.331,E2 -9477.331} C_VEL
LIN {X 0,Y 432.352,Z 296.63,A -85,B 0,C 180,E1 -9480.511,E2 -9480.511} C_VEL
LIN {X 0,Y 432.364,Z 296.629,A -85,B 0,C 180,E1 -9484.004,E2 -9484.004} C_VEL
LIN {X 0,Y 432.325,Z 296.628,A -85,B 0,C 180,E1 -9487.197,E2 -9487.197} C_VEL
LIN {X 0,Y 432.327,Z 296.632,A -85,B 0,C 180,E1 -9490.561,E2 -9490.561} C_VEL
LIN {X 0,Y 432.318,Z 296.629,A -85,B 0,C 180,E1 -9493.061,E2 -9493.061} C_VEL
LIN {X 0,Y 432.335,Z 296.627,A -85,B 0,C 180,E1 -9495.665,E2 -9495.665} C_VEL
LIN {X 0,Y 432.333,Z 296.634,A -85,B 0,C 180,E1 -9498.398,E2 -9498.398} C_VEL
LIN {X 0,Y 432.338,Z 296.627,A -85,B 0,C 180,E1 -9501.85,E2 -9501.85} C_VEL
LIN {X 0,Y 432.339,Z 296.627,A -85,B 0,C 180,E1 -9505.323,E2 -9505.323} C_VEL
LIN {X 0,Y 432.319,Z 296.636,A -85,B 0,C 180,E1 -9508.654,E2 -9508.654} C_VEL
LIN {X 0,Y 432.379,Z 296.621,A -85,B 0,C 180,E1 -9511.876,E2 -9511.876} C_VEL
LIN {X 0,Y 432.348,Z 296.632,A -85,B 0,C 180,E1 -9514.998,E2 -9514.998} C_VEL
LIN {X 0,Y 432.352,Z 296.624,A -85,B 0,C 180,E1 -9518.045,E2 -9518.045} C_VEL
LIN {X 0,Y 432.38,Z 296.629,A -85,B 0,C 180,E1 -9521.029,E2 -9521.029} C_VEL
LIN {X 0,Y 432.424,Z 296.616,A -85,B 0,C 180,E1 -9523.961,E2 -9523.961} C_VEL
LIN {X 0,Y 432.452,Z 296.613,A -85,B 0,C 180,E1 -9527.803,E2 -9527.803} C_VEL
LIN {X 0,Y 432.485,Z 296.612,A -85,B 0,C 180,E1 -9531.59,E2 -9531.59} C_VEL
LIN {X 0,Y 432.583,Z 296.596,A -85,B 0,C 180,E1 -9534.406,E2 -9534.406} C_VEL
LIN {X 0,Y 432.593,Z 296.595,A -85,B 0,C 180,E1 -9538.138,E2 -9538.138} C_VEL
LIN {X 0,Y 432.718,Z 296.581,A -85,B 0,C 180,E1 -9540,E2 -9540} C_VEL
LIN {X 0,Y 432.581,Z 296.596,A -85,B 0,C 180,E1 -9542.794,E2 -9542.794} C_VEL
LIN {X 0,Y 432.571,Z 296.605,A -85,B 0,C 180,E1 -9545.594,E2 -9545.594} C_VEL
LIN {X 0,Y 432.456,Z 296.612,A -85,B 0,C 180,E1 -9548.41,E2 -9548.41} C_VEL
LIN {X 0,Y 432.451,Z 296.615,A -85,B 0,C 180,E1 -9552.197,E2 -9552.197} C_VEL
LIN {X 0,Y 432.422,Z 296.622,A -85,B 0,C 180,E1 -9556.039,E2 -9556.039} C_VEL
LIN {X 0,Y 432.381,Z 296.623,A -85,B 0,C 180,E1 -9559.485,E2 -9559.485} C_VEL
LIN {X 0,Y 432.303,Z 296.63,A -85,B 0,C 180,E1 -9562.965,E2 -9562.965} C_VEL
LIN {X 0,Y 432.312,Z 296.637,A -85,B 0,C 180,E1 -9566.036,E2 -9566.036} C_VEL
LIN {X 0,Y 432.318,Z 296.629,A -85,B 0,C 180,E1 -9569.189,E2 -9569.189} C_VEL
LIN {X 0,Y 432.315,Z 296.635,A -85,B 0,C 180,E1 -9572.444,E2 -9572.444} C_VEL
LIN {X 0,Y 432.33,Z 296.629,A -85,B 0,C 180,E1 -9575.819,E2 -9575.819} C_VEL
LIN {X 0,Y 432.31,Z 296.634,A -85,B 0,C 180,E1 -9578.71,E2 -9578.71} C_VEL
LIN {X 0,Y 432.299,Z 296.632,A -85,B 0,C 180,E1 -9581.801,E2 -9581.801} C_VEL
LIN {X 0,Y 432.332,Z 296.632,A -85,B 0,C 180,E1 -9584.348,E2 -9584.348} C_VEL
LIN {X 0,Y 432.281,Z 296.636,A -85,B 0,C 180,E1 -9587.022,E2 -9587.022} C_VEL
LIN {X 0,Y 432.289,Z 296.632,A -85,B 0,C 180,E1 -9589.828,E2 -9589.828} C_VEL
LIN {X 0,Y 432.285,Z 296.637,A -85,B 0,C 180,E1 -9593.019,E2 -9593.019} C_VEL
LIN {X 0,Y 432.274,Z 296.637,A -85,B 0,C 180,E1 -9596.441,E2 -9596.441} C_VEL
LIN {X 0,Y 432.332,Z 296.627,A -85,B 0,C 180,E1 -9599.738,E2 -9599.738} C_VEL
LIN {X 0,Y 432.29,Z 296.64,A -85,B 0,C 180,E1 -9602.92,E2 -9602.92} C_VEL
LIN {X 0,Y 432.341,Z 296.626,A -85,B 0,C 180,E1 -9606.02,E2 -9606.02} C_VEL
LIN {X 0,Y 432.355,Z 296.631,A -85,B 0,C 180,E1 -9609.045,E2 -9609.045} C_VEL
LIN {X 0,Y 432.361,Z 296.624,A -85,B 0,C 180,E1 -9612.009,E2 -9612.009} C_VEL
LIN {X 0,Y 432.387,Z 296.624,A -85,B 0,C 180,E1 -9614.924,E2 -9614.924} C_VEL
LIN {X 0,Y 432.464,Z 296.613,A -85,B 0,C 180,E1 -9617.801,E2 -9617.801} C_VEL
LIN {X 0,Y 432.452,Z 296.618,A -85,B 0,C 180,E1 -9621.587,E2 -9621.587} C_VEL
LIN {X 0,Y 432.556,Z 296.599,A -85,B 0,C 180,E1 -9624.403,E2 -9624.403} C_VEL
LIN {X 0,Y 432.598,Z 296.595,A -85,B 0,C 180,E1 -9628.135,E2 -9628.135} C_VEL
LIN {X 0,Y 432.641,Z 296.592,A -85,B 0,C 180,E1 -9629.997,E2 -9629.997} C_VEL
LIN {X 0,Y 432.562,Z 296.598,A -85,B 0,C 180,E1 -9632.791,E2 -9632.791} C_VEL
LIN {X 0,Y 432.44,Z 296.614,A -85,B 0,C 180,E1 -9635.014,E2 -9635.014} C_VEL
LIN {X 0,Y 431.873,Z 296.692,A -85,B 0,C 180,E1 -9635.793,E2 -9635.793} C_VEL
LIN {X 0,Y 429.016,Z 297.044,A -85,B 0,C 180,E1 -9637.056,E2 -9637.056} C_VEL
LIN {X 0,Y 426.537,Z 297.356,A -85,B 0,C 180,E1 -9638.077,E2 -9638.077} C_VEL
LIN {X 0,Y 425.473,Z 297.486,A -85,B 0,C 180,E1 -9638.866,E2 -9638.866} C_VEL
LIN {X 0,Y 425.392,Z 297.496,A -85,B 0,C 180,E1 -9639.133,E2 -9639.133} C_VEL
LIN {X 0,Y 425.429,Z 297.672,A -85,B 0,C 180,E1 -9639.985,E2 -9639.985} C_VEL
LIN {X 0,Y 426.965,Z 306.633,A -85,B 0,C 180,E1 -9642.111,E2 -9642.111} C_VEL
LIN {X 0,Y 426.822,Z 312.44,A -85,B 0,C 180,E1 -9643.409,E2 -9643.409} C_VEL
LIN {X 0,Y 430.633,Z 331.735,A -85,B 0,C 180,E1 -9643.92,E2 -9643.92} C_VEL
LIN {X 0,Y 429.466,Z 419.898,A -85,B 0,C 180,E1 -9645.447,E2 -9645.447} C_VEL
LIN {X 0,Y 429.136,Z 433.555,A -85,B 0,C 180,E1 -9645.886,E2 -9645.886} C_VEL
LIN {X 0,Y 428.674,Z 446.132,A -85,B 0,C 180,E1 -9646.485,E2 -9646.485} C_VEL
LIN {X 0,Y 428.141,Z 457.039,A -85,B 0,C 180,E1 -9647.181,E2 -9647.181} C_VEL
LIN {X 0,Y 427.544,Z 467.575,A -85,B 0,C 180,E1 -9648.034,E2 -9648.034} C_VEL
LIN {X 0,Y 426.804,Z 478.153,A -85,B 0,C 180,E1 -9649.099,E2 -9649.099} C_VEL
LIN {X 0,Y 426.236,Z 487.437,A -85,B 0,C 180,E1 -9650.254,E2 -9650.254} C_VEL
LIN {X 0,Y 425.694,Z 495.895,A -85,B 0,C 180,E1 -9651.547,E2 -9651.547} C_VEL
LIN {X 0,Y 425.123,Z 504.088,A -85,B 0,C 180,E1 -9653.113,E2 -9653.113} C_VEL
LIN {X 0,Y 424.758,Z 509.832,A -85,B 0,C 180,E1 -9654.491,E2 -9654.491} C_VEL
LIN {X 0,Y 424.512,Z 514.849,A -85,B 0,C 180,E1 -9656.017,E2 -9656.017} C_VEL
LIN {X 0,Y 424.269,Z 518.783,A -85,B 0,C 180,E1 -9657.628,E2 -9657.628} C_VEL
LIN {X 0,Y 424.135,Z 520.69,A -85,B 0,C 180,E1 -9658.715,E2 -9658.715} C_VEL
LIN {X 0,Y 424.001,Z 522.672,A -85,B 0,C 180,E1 -9660.467,E2 -9660.467} C_VEL
LIN {X 0,Y 424.008,Z 523.256,A -85,B 0,C 180,E1 -9662.292,E2 -9662.292} C_VEL
LIN {X 0,Y 424.025,Z 522.454,A -85,B 0,C 180,E1 -9664.032,E2 -9664.032} C_VEL
LIN {X 0,Y 424.176,Z 520.399,A -85,B 0,C 180,E1 -9665.721,E2 -9665.721} C_VEL
LIN {X 0,Y 424.414,Z 517.141,A -85,B 0,C 180,E1 -9667.359,E2 -9667.359} C_VEL
LIN {X 0,Y 424.661,Z 512.607,A -85,B 0,C 180,E1 -9668.961,E2 -9668.961} C_VEL
LIN {X 0,Y 425.024,Z 506.964,A -85,B 0,C 180,E1 -9670.479,E2 -9670.479} C_VEL
LIN {X 0,Y 425.512,Z 499.847,A -85,B 0,C 180,E1 -9671.991,E2 -9671.991} C_VEL
LIN {X 0,Y 426.187,Z 490.951,A -85,B 0,C 180,E1 -9673.483,E2 -9673.483} C_VEL
LIN {X 0,Y 426.825,Z 482.046,A -85,B 0,C 180,E1 -9674.686,E2 -9674.686} C_VEL
LIN {X 0,Y 427.549,Z 471.847,A -85,B 0,C 180,E1 -9675.807,E2 -9675.807} C_VEL
LIN {X 0,Y 428.029,Z 463.064,A -85,B 0,C 180,E1 -9676.597,E2 -9676.597} C_VEL
LIN {X 0,Y 428.683,Z 451.351,A -85,B 0,C 180,E1 -9677.445,E2 -9677.445} C_VEL
LIN {X 0,Y 429.257,Z 439.421,A -85,B 0,C 180,E1 -9678.094,E2 -9678.094} C_VEL
LIN {X 0,Y 429.65,Z 426.29,A -85,B 0,C 180,E1 -9678.607,E2 -9678.607} C_VEL
LIN {X 0,Y 429.958,Z 413.474,A -85,B 0,C 180,E1 -9678.911,E2 -9678.911} C_VEL
LIN {X 0,Y 430.88,Z 330.657,A -85,B 0,C 180,E1 -9680.346,E2 -9680.346} C_VEL
LIN {X 0,Y 427.023,Z 312.169,A -85,B 0,C 180,E1 -9680.875,E2 -9680.875} C_VEL
LIN {X 0,Y 427.146,Z 307.263,A -85,B 0,C 180,E1 -9681.848,E2 -9681.848} C_VEL
LIN {X 0,Y 425.276,Z 297.513,A -85,B 0,C 180,E1 -9683.942,E2 -9683.942} C_VEL
LIN {X 0,Y 425.243,Z 297.515,A -85,B 0,C 180,E1 -9686.948,E2 -9686.948} C_VEL
LIN {X 0,Y 425.276,Z 297.515,A -85,B 0,C 180,E1 -9690.279,E2 -9690.279} C_VEL
LIN {X 0,Y 425.311,Z 297.508,A -85,B 0,C 180,E1 -9693.502,E2 -9693.502} C_VEL
LIN {X 0,Y 425.26,Z 297.518,A -85,B 0,C 180,E1 -9696.632,E2 -9696.632} C_VEL
LIN {X 0,Y 425.28,Z 297.516,A -85,B 0,C 180,E1 -9700.363,E2 -9700.363} C_VEL
LIN {X 0,Y 425.339,Z 297.5,A -85,B 0,C 180,E1 -9703.686,E2 -9703.686} C_VEL
LIN {X 0,Y 425.361,Z 297.497,A -85,B 0,C 180,E1 -9707.597,E2 -9707.597} C_VEL
LIN {X 0,Y 425.391,Z 297.493,A -85,B 0,C 180,E1 -9711.449,E2 -9711.449} C_VEL
LIN {X 0,Y 425.499,Z 297.481,A -85,B 0,C 180,E1 -9714.312,E2 -9714.312} C_VEL
LIN {X 0,Y 425.524,Z 297.477,A -85,B 0,C 180,E1 -9718.107,E2 -9718.107} C_VEL
LIN {X 0,Y 425.65,Z 297.455,A -85,B 0,C 180,E1 -9720,E2 -9720} C_VEL
LIN {X 0,Y 425.513,Z 297.48,A -85,B 0,C 180,E1 -9722.84,E2 -9722.84} C_VEL
LIN {X 0,Y 425.481,Z 297.485,A -85,B 0,C 180,E1 -9726.64,E2 -9726.64} C_VEL
LIN {X 0,Y 425.357,Z 297.5,A -85,B 0,C 180,E1 -9729.51,E2 -9729.51} C_VEL
LIN {X 0,Y 425.355,Z 297.496,A -85,B 0,C 180,E1 -9732.912,E2 -9732.912} C_VEL
LIN {X 0,Y 425.321,Z 297.497,A -85,B 0,C 180,E1 -9736.61,E2 -9736.61} C_VEL
LIN {X 0,Y 425.315,Z 297.499,A -85,B 0,C 180,E1 -9739.65,E2 -9739.65} C_VEL
LIN {X 0,Y 425.273,Z 297.508,A -85,B 0,C 180,E1 -9743.367,E2 -9743.367} C_VEL
LIN {X 0,Y 425.305,Z 297.504,A -85,B 0,C 180,E1 -9746.847,E2 -9746.847} C_VEL
LIN {X 0,Y 425.276,Z 297.511,A -85,B 0,C 180,E1 -9749.721,E2 -9749.721} C_VEL
LIN {X 0,Y 425.243,Z 297.512,A -85,B 0,C 180,E1 -9753.052,E2 -9753.052} C_VEL
LIN {X 0,Y 425.25,Z 297.514,A -85,B 0,C 180,E1 -9755.933,E2 -9755.933} C_VEL
LIN {X 0,Y 425.304,Z 297.504,A -85,B 0,C 180,E1 -9759.054,E2 -9759.054} C_VEL
LIN {X 0,Y 425.3,Z 297.508,A -85,B 0,C 180,E1 -9762.65,E2 -9762.65} C_VEL
LIN {X 0,Y 425.306,Z 297.51,A -85,B 0,C 180,E1 -9766.058,E2 -9766.058} C_VEL
LIN {X 0,Y 425.283,Z 297.51,A -85,B 0,C 180,E1 -9768.63,E2 -9768.63} C_VEL
LIN {X 0,Y 425.301,Z 297.507,A -85,B 0,C 180,E1 -9771.109,E2 -9771.109} C_VEL
LIN {X 0,Y 425.279,Z 297.511,A -85,B 0,C 180,E1 -9774.669,E2 -9774.669} C_VEL
LIN {X 0,Y 425.248,Z 297.52,A -85,B 0,C 180,E1 -9778.078,E2 -9778.078} C_VEL
LIN {X 0,Y 425.322,Z 297.509,A -85,B 0,C 180,E1 -9781.373,E2 -9781.373} C_VEL
LIN {X 0,Y 425.365,Z 297.549,A -85,B 0,C 180,E1 -9782.681,E2 -9782.681} C_VEL
LIN {X 0,Y 428.118,Z 311.269,A -85,B 0,C 180,E1 -9785.517,E2 -9785.517} C_VEL
LIN {X 0,Y 427.739,Z 320.949,A -85,B 0,C 180,E1 -9787.348,E2 -9787.348} C_VEL
LIN {X 0,Y 426.613,Z 341.169,A -85,B 0,C 180,E1 -9791.111,E2 -9791.111} C_VEL
LIN {X 0,Y 426.979,Z 343.551,A -85,B 0,C 180,E1 -9791.214,E2 -9791.214} C_VEL
LIN {X 0,Y 430.617,Z 367.764,A -85,B 0,C 180,E1 -9791.818,E2 -9791.818} C_VEL
LIN {X 0,Y 429.572,Z 450.884,A -85,B 0,C 180,E1 -9793.276,E2 -9793.276} C_VEL
LIN {X 0,Y 429.04,Z 464.58,A -85,B 0,C 180,E1 -9793.713,E2 -9793.713} C_VEL
LIN {X 0,Y 428.446,Z 476.947,A -85,B 0,C 180,E1 -9794.301,E2 -9794.301} C_VEL
LIN {X 0,Y 427.779,Z 488.033,A -85,B 0,C 180,E1 -9795.008,E2 -9795.008} C_VEL
LIN {X 0,Y 427.117,Z 499.303,A -85,B 0,C 180,E1 -9795.929,E2 -9795.929} C_VEL
LIN {X 0,Y 426.358,Z 510.072,A -85,B 0,C 180,E1 -9797.025,E2 -9797.025} C_VEL
LIN {X 0,Y 425.811,Z 518.636,A -85,B 0,C 180,E1 -9798.098,E2 -9798.098} C_VEL
LIN {X 0,Y 425.113,Z 527.921,A -85,B 0,C 180,E1 -9799.526,E2 -9799.526} C_VEL
LIN {X 0,Y 424.715,Z 535.397,A -85,B 0,C 180,E1 -9800.959,E2 -9800.959} C_VEL
LIN {X 0,Y 424.411,Z 541.404,A -85,B 0,C 180,E1 -9802.391,E2 -9802.391} C_VEL
LIN {X 0,Y 424.239,Z 545.799,A -85,B 0,C 180,E1 -9803.706,E2 -9803.706} C_VEL
LIN {X 0,Y 424.198,Z 549.783,A -85,B 0,C 180,E1 -9805.252,E2 -9805.252} C_VEL
LIN {X 0,Y 424.099,Z 551.646,A -85,B 0,C 180,E1 -9806.203,E2 -9806.203} C_VEL
LIN {X 0,Y 424.133,Z 553.049,A -85,B 0,C 180,E1 -9807.154,E2 -9807.154} C_VEL
LIN {X 0,Y 424.143,Z 554.052,A -85,B 0,C 180,E1 -9808.104,E2 -9808.104} C_VEL
LIN {X 0,Y 424.111,Z 554.662,A -85,B 0,C 180,E1 -9809.054,E2 -9809.054} C_VEL
LIN {X 0,Y 424.109,Z 554.863,A -85,B 0,C 180,E1 -9810.003,E2 -9810.003} C_VEL
LIN {X 0,Y 424.144,Z 554.012,A -85,B 0,C 180,E1 -9811.902,E2 -9811.902} C_VEL
LIN {X 0,Y 424.135,Z 552.998,A -85,B 0,C 180,E1 -9812.852,E2 -9812.852} C_VEL
LIN {X 0,Y 424.102,Z 551.559,A -85,B 0,C 180,E1 -9813.804,E2 -9813.804} C_VEL
LIN {X 0,Y 424.208,Z 548.573,A -85,B 0,C 180,E1 -9815.231,E2 -9815.231} C_VEL
LIN {X 0,Y 424.302,Z 544.524,A -85,B 0,C 180,E1 -9816.661,E2 -9816.661} C_VEL
LIN {X 0,Y 424.541,Z 538.287,A -85,B 0,C 180,E1 -9818.331,E2 -9818.331} C_VEL
LIN {X 0,Y 424.893,Z 531.49,A -85,B 0,C 180,E1 -9819.764,E2 -9819.764} C_VEL
LIN {X 0,Y 425.416,Z 523.044,A -85,B 0,C 180,E1 -9821.195,E2 -9821.195} C_VEL
LIN {X 0,Y 426.028,Z 514.338,A -85,B 0,C 180,E1 -9822.386,E2 -9822.386} C_VEL
LIN {X 0,Y 426.717,Z 503.627,A -85,B 0,C 180,E1 -9823.575,E2 -9823.575} C_VEL
LIN {X 0,Y 427.329,Z 492.964,A -85,B 0,C 180,E1 -9824.527,E2 -9824.527} C_VEL
LIN {X 0,Y 428.065,Z 481.081,A -85,B 0,C 180,E1 -9825.354,E2 -9825.354} C_VEL
LIN {X 0,Y 428.644,Z 468.731,A -85,B 0,C 180,E1 -9826.003,E2 -9826.003} C_VEL
LIN {X 0,Y 429.188,Z 456.107,A -85,B 0,C 180,E1 -9826.471,E2 -9826.471} C_VEL
LIN {X 0,Y 429.542,Z 441.31,A -85,B 0,C 180,E1 -9826.793,E2 -9826.793} C_VEL
LIN {X 0,Y 430.303,Z 367.071,A -85,B 0,C 180,E1 -9828.066,E2 -9828.066} C_VEL
LIN {X 0,Y 426.54,Z 342.131,A -85,B 0,C 180,E1 -9828.693,E2 -9828.693} C_VEL
LIN {X 0,Y 427.579,Z 324.984,A -85,B 0,C 180,E1 -9831.96,E2 -9831.96} C_VEL
LIN {X 0,Y 428.289,Z 313.266,A -85,B 0,C 180,E1 -9834.221,E2 -9834.221} C_VEL
LIN {X 0,Y 426.716,Z 304.035,A -85,B 0,C 180,E1 -9836.142,E2 -9836.142} C_VEL
LIN {X 0,Y 425.403,Z 297.496,A -85,B 0,C 180,E1 -9837.555,E2 -9837.555} C_VEL
LIN {X 0,Y 425.293,Z 297.508,A -85,B 0,C 180,E1 -9840.817,E2 -9840.817} C_VEL
LIN {X 0,Y 425.316,Z 297.507,A -85,B 0,C 180,E1 -9844.288,E2 -9844.288} C_VEL
LIN {X 0,Y 425.281,Z 297.507,A -85,B 0,C 180,E1 -9847.695,E2 -9847.695} C_VEL
LIN {X 0,Y 425.282,Z 297.51,A -85,B 0,C 180,E1 -9850.52,E2 -9850.52} C_VEL
LIN {X 0,Y 425.259,Z 297.508,A -85,B 0,C 180,E1 -9853.351,E2 -9853.351} C_VEL
LIN {X 0,Y 425.259,Z 297.514,A -85,B 0,C 180,E1 -9856.649,E2 -9856.649} C_VEL
LIN {X 0,Y 425.289,Z 297.505,A -85,B 0,C 180,E1 -9859.873,E2 -9859.873} C_VEL
LIN {X 0,Y 425.278,Z 297.512,A -85,B 0,C 180,E1 -9862.488,E2 -9862.488} C_VEL
LIN {X 0,Y 425.306,Z 297.502,A -85,B 0,C 180,E1 -9865.817,E2 -9865.817} C_VEL
LIN {X 0,Y 425.289,Z 297.507,A -85,B 0,C 180,E1 -9869.239,E2 -9869.239} C_VEL
LIN {X 0,Y 425.346,Z 297.5,A -85,B 0,C 180,E1 -9872.442,E2 -9872.442} C_VEL
LIN {X 0,Y 425.347,Z 297.498,A -85,B 0,C 180,E1 -9875.602,E2 -9875.602} C_VEL
LIN {X 0,Y 425.287,Z 297.509,A -85,B 0,C 180,E1 -9878.681,E2 -9878.681} C_VEL
LIN {X 0,Y 425.326,Z 297.501,A -85,B 0,C 180,E1 -9881.702,E2 -9881.702} C_VEL
LIN {X 0,Y 425.34,Z 297.5,A -85,B 0,C 180,E1 -9884.67,E2 -9884.67} C_VEL
LIN {X 0,Y 425.405,Z 297.493,A -85,B 0,C 180,E1 -9887.598,E2 -9887.598} C_VEL
LIN {X 0,Y 425.436,Z 297.492,A -85,B 0,C 180,E1 -9891.45,E2 -9891.45} C_VEL
LIN {X 0,Y 425.54,Z 297.473,A -85,B 0,C 180,E1 -9894.313,E2 -9894.313} C_VEL
LIN {X 0,Y 425.563,Z 297.471,A -85,B 0,C 180,E1 -9898.107,E2 -9898.107} C_VEL
LIN {X 0,Y 425.688,Z 297.457,A -85,B 0,C 180,E1 -9900,E2 -9900} C_VEL
LIN {X 0,Y 425.535,Z 297.474,A -85,B 0,C 180,E1 -9902.84,E2 -9902.84} C_VEL
LIN {X 0,Y 425.474,Z 297.481,A -85,B 0,C 180,E1 -9906.531,E2 -9906.531} C_VEL
LIN {X 0,Y 425.39,Z 297.497,A -85,B 0,C 180,E1 -9909.51,E2 -9909.51} C_VEL
LIN {X 0,Y 425.387,Z 297.492,A -85,B 0,C 180,E1 -9912.903,E2 -9912.903} C_VEL
LIN {X 0,Y 425.354,Z 297.497,A -85,B 0,C 180,E1 -9916.604,E2 -9916.604} C_VEL
LIN {X 0,Y 425.323,Z 297.504,A -85,B 0,C 180,E1 -9919.635,E2 -9919.635} C_VEL
LIN {X 0,Y 425.282,Z 297.509,A -85,B 0,C 180,E1 -9922.339,E2 -9922.339} C_VEL
LIN {X 0,Y 425.254,Z 297.51,A -85,B 0,C 180,E1 -9925.448,E2 -9925.448} C_VEL
LIN {X 0,Y 425.296,Z 297.504,A -85,B 0,C 180,E1 -9928.858,E2 -9928.858} C_VEL
LIN {X 0,Y 425.256,Z 297.512,A -85,B 0,C 180,E1 -9931.928,E2 -9931.928} C_VEL
LIN {X 0,Y 425.289,Z 297.504,A -85,B 0,C 180,E1 -9935.337,E2 -9935.337} C_VEL
LIN {X 0,Y 425.263,Z 297.51,A -85,B 0,C 180,E1 -9938.903,E2 -9938.903} C_VEL
LIN {X 0,Y 425.242,Z 297.512,A -85,B 0,C 180,E1 -9941.951,E2 -9941.951} C_VEL
LIN {X 0,Y 425.271,Z 297.507,A -85,B 0,C 180,E1 -9945.285,E2 -9945.285} C_VEL
LIN {X 0,Y 425.246,Z 297.518,A -85,B 0,C 180,E1 -9948.617,E2 -9948.617} C_VEL
LIN {X 0,Y 425.266,Z 297.51,A -85,B 0,C 180,E1 -9952.304,E2 -9952.304} C_VEL
LIN {X 0,Y 425.237,Z 297.511,A -85,B 0,C 180,E1 -9955.81,E2 -9955.81} C_VEL
LIN {X 0,Y 425.288,Z 297.508,A -85,B 0,C 180,E1 -9959.24,E2 -9959.24} C_VEL
LIN {X 0,Y 425.239,Z 297.512,A -85,B 0,C 180,E1 -9962.433,E2 -9962.433} C_VEL
LIN {X 0,Y 425.322,Z 297.502,A -85,B 0,C 180,E1 -9965.599,E2 -9965.599} C_VEL
LIN {X 0,Y 425.298,Z 297.506,A -85,B 0,C 180,E1 -9968.68,E2 -9968.68} C_VEL
LIN {X 0,Y 425.324,Z 297.502,A -85,B 0,C 180,E1 -9971.7,E2 -9971.7} C_VEL
LIN {X 0,Y 425.341,Z 297.499,A -85,B 0,C 180,E1 -9974.668,E2 -9974.668} C_VEL
LIN {X 0,Y 425.417,Z 297.493,A -85,B 0,C 180,E1 -9977.596,E2 -9977.596} C_VEL
LIN {X 0,Y 425.4,Z 297.499,A -85,B 0,C 180,E1 -9981.447,E2 -9981.447} C_VEL
LIN {X 0,Y 425.514,Z 297.477,A -85,B 0,C 180,E1 -9984.31,E2 -9984.31} C_VEL
LIN {X 0,Y 425.567,Z 297.472,A -85,B 0,C 180,E1 -9988.104,E2 -9988.104} C_VEL
LIN {X 0,Y 425.593,Z 297.47,A -85,B 0,C 180,E1 -9989.997,E2 -9989.997} C_VEL
LIN {X 0,Y 425.517,Z 297.476,A -85,B 0,C 180,E1 -9992.837,E2 -9992.837} C_VEL
LIN {X 0,Y 425.527,Z 297.482,A -85,B 0,C 180,E1 -9995.684,E2 -9995.684} C_VEL
LIN {X 0,Y 425.406,Z 297.495,A -85,B 0,C 180,E1 -9998.547,E2 -9998.547} C_VEL
LIN {X 0,Y 425.392,Z 297.496,A -85,B 0,C 180,E1 -9999.133,E2 -9999.133} C_VEL
LIN {X 0,Y 425.161,Z 298.001,A -85,B 0,C 180,E1 -9999.657,E2 -9999.657} C_VEL
LIN {X 0,Y 424.568,Z 299.278,A -85,B 0,C 180,E1 -10000.154,E2 -10000.154} C_VEL
LIN {X 0,Y 422.793,Z 303.111,A -85,B 0,C 180,E1 -10001.082,E2 -10001.082} C_VEL
LIN {X 0,Y 420.281,Z 309.637,A -85,B 0,C 180,E1 -10002.433,E2 -10002.433} C_VEL
LIN {X 0,Y 419.967,Z 311.749,A -85,B 0,C 180,E1 -10002.899,E2 -10002.899} C_VEL
LIN {X 0,Y 419.95,Z 312.847,A -85,B 0,C 180,E1 -10003.115,E2 -10003.115} C_VEL
LIN {X 0,Y 423.87,Z 332.579,A -85,B 0,C 180,E1 -10003.647,E2 -10003.647} C_VEL
LIN {X 0,Y 422.644,Z 420.563,A -85,B 0,C 180,E1 -10005.201,E2 -10005.201} C_VEL
LIN {X 0,Y 422.285,Z 434.32,A -85,B 0,C 180,E1 -10005.655,E2 -10005.655} C_VEL
LIN {X 0,Y 421.803,Z 446.737,A -85,B 0,C 180,E1 -10006.263,E2 -10006.263} C_VEL
LIN {X 0,Y 421.108,Z 459.308,A -85,B 0,C 180,E1 -10007.102,E2 -10007.102} C_VEL
LIN {X 0,Y 420.462,Z 470.657,A -85,B 0,C 180,E1 -10008.08,E2 -10008.08} C_VEL
LIN {X 0,Y 419.734,Z 480.824,A -85,B 0,C 180,E1 -10009.179,E2 -10009.179} C_VEL
LIN {X 0,Y 419.025,Z 490.415,A -85,B 0,C 180,E1 -10010.465,E2 -10010.465} C_VEL
LIN {X 0,Y 418.51,Z 498.864,A -85,B 0,C 180,E1 -10011.868,E2 -10011.868} C_VEL
LIN {X 0,Y 418.045,Z 505.66,A -85,B 0,C 180,E1 -10013.265,E2 -10013.265} C_VEL
LIN {X 0,Y 417.607,Z 511.844,A -85,B 0,C 180,E1 -10014.875,E2 -10014.875} C_VEL
LIN {X 0,Y 417.366,Z 516.296,A -85,B 0,C 180,E1 -10016.375,E2 -10016.375} C_VEL
LIN {X 0,Y 417.109,Z 520.121,A -85,B 0,C 180,E1 -10018.144,E2 -10018.144} C_VEL
LIN {X 0,Y 416.994,Z 521.753,A -85,B 0,C 180,E1 -10019.254,E2 -10019.254} C_VEL
LIN {X 0,Y 416.91,Z 523.102,A -85,B 0,C 180,E1 -10020.714,E2 -10020.714} C_VEL
LIN {X 0,Y 416.927,Z 523.472,A -85,B 0,C 180,E1 -10022.637,E2 -10022.637} C_VEL
LIN {X 0,Y 416.947,Z 522.526,A -85,B 0,C 180,E1 -10024.316,E2 -10024.316} C_VEL
LIN {X 0,Y 417.165,Z 520.116,A -85,B 0,C 180,E1 -10026.125,E2 -10026.125} C_VEL
LIN {X 0,Y 417.383,Z 516.847,A -85,B 0,C 180,E1 -10027.683,E2 -10027.683} C_VEL
LIN {X 0,Y 417.645,Z 512.252,A -85,B 0,C 180,E1 -10029.279,E2 -10029.279} C_VEL
LIN {X 0,Y 418.063,Z 505.896,A -85,B 0,C 180,E1 -10030.959,E2 -10030.959} C_VEL
LIN {X 0,Y 418.672,Z 497.885,A -85,B 0,C 180,E1 -10032.586,E2 -10032.586} C_VEL
LIN {X 0,Y 419.409,Z 489.116,A -85,B 0,C 180,E1 -10034.003,E2 -10034.003} C_VEL
LIN {X 0,Y 420.114,Z 479.872,A -85,B 0,C 180,E1 -10035.21,E2 -10035.21} C_VEL
LIN {X 0,Y 420.734,Z 470.093,A -85,B 0,C 180,E1 -10036.249,E2 -10036.249} C_VEL
LIN {X 0,Y 421.574,Z 458.092,A -85,B 0,C 180,E1 -10037.261,E2 -10037.261} C_VEL
LIN {X 0,Y 422.136,Z 447.301,A -85,B 0,C 180,E1 -10037.974,E2 -10037.974} C_VEL
LIN {X 0,Y 422.607,Z 435,A -85,B 0,C 180,E1 -10038.584,E2 -10038.584} C_VEL
LIN {X 0,Y 423.036,Z 421.793,A -85,B 0,C 180,E1 -10039.027,E2 -10039.027} C_VEL
LIN {X 0,Y 423.511,Z 387.99,A -85,B 0,C 180,E1 -10039.653,E2 -10039.653} C_VEL
LIN {X 0,Y 424.26,Z 332.116,A -85,B 0,C 180,E1 -10040.636,E2 -10040.636} C_VEL
LIN {X 0,Y 420.149,Z 312.393,A -85,B 0,C 180,E1 -10041.227,E2 -10041.227} C_VEL
LIN {X 0,Y 420.168,Z 308.135,A -85,B 0,C 180,E1 -10042.091,E2 -10042.091} C_VEL
LIN {X 0,Y 418.241,Z 298.391,A -85,B 0,C 180,E1 -10044.198,E2 -10044.198} C_VEL
LIN {X 0,Y 418.206,Z 298.391,A -85,B 0,C 180,E1 -10047.468,E2 -10047.468} C_VEL
LIN {X 0,Y 418.235,Z 298.389,A -85,B 0,C 180,E1 -10050.89,E2 -10050.89} C_VEL
LIN {X 0,Y 418.227,Z 298.395,A -85,B 0,C 180,E1 -10054.093,E2 -10054.093} C_VEL
LIN {X 0,Y 418.192,Z 298.395,A -85,B 0,C 180,E1 -10057.261,E2 -10057.261} C_VEL
LIN {X 0,Y 418.235,Z 298.394,A -85,B 0,C 180,E1 -10060.362,E2 -10060.362} C_VEL
LIN {X 0,Y 418.268,Z 298.381,A -85,B 0,C 180,E1 -10063.403,E2 -10063.403} C_VEL
LIN {X 0,Y 418.296,Z 298.38,A -85,B 0,C 180,E1 -10066.998,E2 -10066.998} C_VEL
LIN {X 0,Y 418.29,Z 298.378,A -85,B 0,C 180,E1 -10070.327,E2 -10070.327} C_VEL
LIN {X 0,Y 418.439,Z 298.36,A -85,B 0,C 180,E1 -10073.248,E2 -10073.248} C_VEL
LIN {X 0,Y 418.288,Z 298.377,A -85,B 0,C 180,E1 -10075.181,E2 -10075.181} C_VEL
LIN {X 0,Y 418.494,Z 298.352,A -85,B 0,C 180,E1 -10078.075,E2 -10078.075} C_VEL
LIN {X 0,Y 418.62,Z 298.33,A -85,B 0,C 180,E1 -10080,E2 -10080} C_VEL
LIN {X 0,Y 418.467,Z 298.357,A -85,B 0,C 180,E1 -10082.888,E2 -10082.888} C_VEL
LIN {X 0,Y 418.443,Z 298.363,A -85,B 0,C 180,E1 -10086.752,E2 -10086.752} C_VEL
LIN {X 0,Y 418.313,Z 298.376,A -85,B 0,C 180,E1 -10089.672,E2 -10089.672} C_VEL
LIN {X 0,Y 418.306,Z 298.375,A -85,B 0,C 180,E1 -10093.008,E2 -10093.008} C_VEL
LIN {X 0,Y 418.272,Z 298.376,A -85,B 0,C 180,E1 -10096.74,E2 -10096.74} C_VEL
LIN {X 0,Y 418.257,Z 298.377,A -85,B 0,C 180,E1 -10099.805,E2 -10099.805} C_VEL
LIN {X 0,Y 418.232,Z 298.384,A -85,B 0,C 180,E1 -10102.737,E2 -10102.737} C_VEL
LIN {X 0,Y 418.231,Z 298.385,A -85,B 0,C 180,E1 -10105.907,E2 -10105.907} C_VEL
LIN {X 0,Y 418.232,Z 298.384,A -85,B 0,C 180,E1 -10109.165,E2 -10109.165} C_VEL
LIN {X 0,Y 418.218,Z 298.386,A -85,B 0,C 180,E1 -10112.847,E2 -10112.847} C_VEL
LIN {X 0,Y 418.215,Z 298.388,A -85,B 0,C 180,E1 -10116.243,E2 -10116.243} C_VEL
LIN {X 0,Y 418.243,Z 298.391,A -85,B 0,C 180,E1 -10119.683,E2 -10119.683} C_VEL
LIN {X 0,Y 418.253,Z 298.387,A -85,B 0,C 180,E1 -10122.334,E2 -10122.334} C_VEL
LIN {X 0,Y 418.245,Z 298.389,A -85,B 0,C 180,E1 -10125.118,E2 -10125.118} C_VEL
LIN {X 0,Y 418.265,Z 298.389,A -85,B 0,C 180,E1 -10127.778,E2 -10127.778} C_VEL
LIN {X 0,Y 418.244,Z 298.39,A -85,B 0,C 180,E1 -10131.564,E2 -10131.564} C_VEL
LIN {X 0,Y 418.239,Z 298.388,A -85,B 0,C 180,E1 -10135.164,E2 -10135.164} C_VEL
LIN {X 0,Y 418.227,Z 298.394,A -85,B 0,C 180,E1 -10137.477,E2 -10137.477} C_VEL
LIN {X 0,Y 418.261,Z 298.388,A -85,B 0,C 180,E1 -10140.898,E2 -10140.898} C_VEL
LIN {X 0,Y 418.338,Z 298.511,A -85,B 0,C 180,E1 -10142.421,E2 -10142.421} C_VEL
LIN {X 0,Y 421.164,Z 312.406,A -85,B 0,C 180,E1 -10145.349,E2 -10145.349} C_VEL
LIN {X 0,Y 420.977,Z 319.208,A -85,B 0,C 180,E1 -10146.664,E2 -10146.664} C_VEL
LIN {X 0,Y 419.884,Z 337.967,A -85,B 0,C 180,E1 -10150.22,E2 -10150.22} C_VEL
LIN {X 0,Y 419.731,Z 341.39,A -85,B 0,C 180,E1 -10150.821,E2 -10150.821} C_VEL
LIN {X 0,Y 423.815,Z 367.485,A -85,B 0,C 180,E1 -10151.5,E2 -10151.5} C_VEL
LIN {X 0,Y 422.868,Z 448.682,A -85,B 0,C 180,E1 -10152.94,E2 -10152.94} C_VEL
LIN {X 0,Y 422.39,Z 461.591,A -85,B 0,C 180,E1 -10153.325,E2 -10153.325} C_VEL
LIN {X 0,Y 421.717,Z 474.674,A -85,B 0,C 180,E1 -10153.92,E2 -10153.92} C_VEL
LIN {X 0,Y 421.015,Z 486.271,A -85,B 0,C 180,E1 -10154.637,E2 -10154.637} C_VEL
LIN {X 0,Y 420.297,Z 498.144,A -85,B 0,C 180,E1 -10155.598,E2 -10155.598} C_VEL
LIN {X 0,Y 419.51,Z 508.83,A -85,B 0,C 180,E1 -10156.686,E2 -10156.686} C_VEL
LIN {X 0,Y 418.836,Z 518.445,A -85,B 0,C 180,E1 -10157.896,E2 -10157.896} C_VEL
LIN {X 0,Y 418.094,Z 527.705,A -85,B 0,C 180,E1 -10159.348,E2 -10159.348} C_VEL
LIN {X 0,Y 417.658,Z 535.167,A -85,B 0,C 180,E1 -10160.805,E2 -10160.805} C_VEL
LIN {X 0,Y 417.35,Z 541.166,A -85,B 0,C 180,E1 -10162.261,E2 -10162.261} C_VEL
LIN {X 0,Y 417.163,Z 545.895,A -85,B 0,C 180,E1 -10163.712,E2 -10163.712} C_VEL
LIN {X 0,Y 417.105,Z 549.535,A -85,B 0,C 180,E1 -10165.171,E2 -10165.171} C_VEL
LIN {X 0,Y 417.015,Z 551.394,A -85,B 0,C 180,E1 -10166.138,E2 -10166.138} C_VEL
LIN {X 0,Y 417.031,Z 552.793,A -85,B 0,C 180,E1 -10167.105,E2 -10167.105} C_VEL
LIN {X 0,Y 417.069,Z 553.795,A -85,B 0,C 180,E1 -10168.072,E2 -10168.072} C_VEL
LIN {X 0,Y 417.032,Z 554.402,A -85,B 0,C 180,E1 -10169.038,E2 -10169.038} C_VEL
LIN {X 0,Y 417.028,Z 554.597,A -85,B 0,C 180,E1 -10170.003,E2 -10170.003} C_VEL
LIN {X 0,Y 417.07,Z 553.74,A -85,B 0,C 180,E1 -10171.934,E2 -10171.934} C_VEL
LIN {X 0,Y 417.033,Z 552.72,A -85,B 0,C 180,E1 -10172.901,E2 -10172.901} C_VEL
LIN {X 0,Y 417.017,Z 551.273,A -85,B 0,C 180,E1 -10173.868,E2 -10173.868} C_VEL
LIN {X 0,Y 417.122,Z 548.279,A -85,B 0,C 180,E1 -10175.32,E2 -10175.32} C_VEL
LIN {X 0,Y 417.234,Z 544.219,A -85,B 0,C 180,E1 -10176.774,E2 -10176.774} C_VEL
LIN {X 0,Y 417.498,Z 537.967,A -85,B 0,C 180,E1 -10178.473,E2 -10178.473} C_VEL
LIN {X 0,Y 417.874,Z 531.156,A -85,B 0,C 180,E1 -10179.929,E2 -10179.929} C_VEL
LIN {X 0,Y 418.426,Z 522.687,A -85,B 0,C 180,E1 -10181.385,E2 -10181.385} C_VEL
LIN {X 0,Y 419.055,Z 513.957,A -85,B 0,C 180,E1 -10182.595,E2 -10182.595} C_VEL
LIN {X 0,Y 419.786,Z 503.02,A -85,B 0,C 180,E1 -10183.824,E2 -10183.824} C_VEL
LIN {X 0,Y 420.43,Z 492.524,A -85,B 0,C 180,E1 -10184.771,E2 -10184.771} C_VEL
LIN {X 0,Y 421.174,Z 480.573,A -85,B 0,C 180,E1 -10185.611,E2 -10185.611} C_VEL
LIN {X 0,Y 421.812,Z 468.149,A -85,B 0,C 180,E1 -10186.269,E2 -10186.269} C_VEL
LIN {X 0,Y 422.38,Z 455.362,A -85,B 0,C 180,E1 -10186.744,E2 -10186.744} C_VEL
LIN {X 0,Y 422.741,Z 440.193,A -85,B 0,C 180,E1 -10187.072,E2 -10187.072} C_VEL
LIN {X 0,Y 423.442,Z 367.163,A -85,B 0,C 180,E1 -10188.349,E2 -10188.349} C_VEL
LIN {X 0,Y 419.591,Z 341.966,A -85,B 0,C 180,E1 -10188.983,E2 -10188.983} C_VEL
